			CNC_ZeroOffsets:
				IF (nLogChannelID <= 0 OR nLogChannelID > nLogChannelID) THEN
					nErrorID 	:= ErrID_7;
					Step := 999;
				ELSE
					Step := 12;
				END_IF
		END_CASE
	END_IF

	fbFileOpen.bExecute := FALSE;
	
	// Check Channel State
	IF (CNCSystem.LogChannelNo[nLogChannelID].nHliChannelIdx <> -1) THEN
		
		IF (cncSystem.Channel[CNCSystem.LogChannelNo[nLogChannelID].nHliChannelIdx].ActState <> HLI_IMCM_PROCESS_SELECTED AND 
			cncSystem.Channel[CNCSystem.LogChannelNo[nLogChannelID].nHliChannelIdx].ActState <> HLI_IMCM_PROCESS_READY) THEN
			nErrorID 	:= ErrID_10;
			Step := 999;
		END_IF				
	ELSE
			nErrorID 	:= ErrID_7;
			Step := 999;		
	END_IF			

12:	(* create file name and list file header  *)
	strHeader := '';

	CASE eParameterType OF

		CNC_AxisParameter:
			strFileName := CONCAT(strTempPath, '\axis');
			strFileName := CONCAT(strFileName, UINT_TO_STRING(nLogAxisId));
			strFileName := CONCAT(strFileName, '.lis');

			strHeader := 'kopf.achs_nr ';
			strHeader := CONCAT(strHeader, UINT_TO_STRING(nLogAxisId));
			Step := 15;
		CNC_ChannelParameter:
			strFileName := CONCAT(strTempPath, '\channel');			
			strFileName := CONCAT(strFileName, UINT_TO_STRING(nLogChannelID));
			strFileName := CONCAT(strFileName, '.lis');
			Step := 15;
		CNC_ToolParameter:			
			strFileName := CONCAT(strTempPath, '\ToolCh');
			strFileName := CONCAT(strFileName, UINT_TO_STRING(nLogChannelID));
			strFileName := CONCAT(strFileName, '.lis');
			Step := 15;
		CNC_ClampPosition:
			strFileName := CONCAT(strTempPath, '\ClampPosCh');			
			strFileName := CONCAT(strFileName, UINT_TO_STRING(nLogChannelID));
			strFileName := CONCAT(strFileName, '.lis');
			Step := 15;
		CNC_ZeroOffsets:			
			strFileName := CONCAT(strTempPath, '\ZeroOffsetsChh');
			strFileName := CONCAT(strFileName, UINT_TO_STRING(nLogChannelID));
			strFileName := CONCAT(strFileName, '.lis');
			Step := 15;
		ELSE
			nErrorID 	:= ErrID_5;
			Step := 999;
	END_CASE

15:	(* write file to destination folder *)
	fbFileOpen.sNetId := '';
	fbFileOpen.sPathName := strFileName;
	fbFileOpen.nMode := FOPEN_MODEWRITE OR FOPEN_MODETEXT;
	fbFileOpen.ePath := PATH_GENERIC;
	fbFileOpen.tTimeout := t#1s;
	fbFileOpen.bExecute := TRUE;
	Step := 16;

16:
	IF ( NOT fbFileOpen.bBusy ) THEN
		IF ( fbFileOpen.bError ) THEN
			nErrorID  :=ErrID_9 ;
			bError := TRUE;
			Step := 999;
		ELSE
			hFileOutput := fbFileOpen.hFile;
			fbFilePuts.bExecute:= FALSE;
			Step := 17;
		END_IF
	END_IF


17: (* Write Header File *)
	fbFilePuts.sNetId:='';
	fbFilePuts.hFile:=hFileOutput;
	fbFilePuts.bExecute:=TRUE;
	fbFilePuts.tTimeout:=t#10s;
	fbFilePuts.sLine :=strHeader;
	Step := 18;

18:
	IF ( NOT fbFilePuts.bBusy ) THEN
		IF ( fbFilePuts.bError ) THEN
			 nErrorID  :=ErrID_9 ;
			bError := TRUE;
			Step := 999;
		ELSE
			fbFilePuts.bExecute:= FALSE;
			m := 0;
			Step := 19;
		END_IF
	END_IF


19:	(* Write Parameter lines *)
		strParameterLine :=  CONCAT('$N',stParameter[m].strName);
		strParameterLine :=  CONCAT(strParameterLine,'   ');
		strParameterLine := CONCAT(strParameterLine, stParameter[m].strValue);
		fbFilePuts.sLine :=strParameterLine;
		fbFilePuts.bExecute:= TRUE;
		Step := 20;
20:
		IF ( NOT fbFilePuts.bBusy ) THEN
			IF ( fbFilePuts.bError ) THEN
				 nErrorID  :=ErrID_9 ;
				bError := TRUE;
				Step := 999;
			ELSE
				Step := 21;
			END_IF
		END_IF

21:	(* Next Line *)
	IF (m+1 <= (nMaxParameters-1) AND m+1 <= nNumParameters) THEN
		m := m+1;
		fbFilePuts.bExecute:= FALSE;
		Step := 19;
	ELSE
		fbFilePuts.bExecute:= FALSE;
		Step := 22;
	END_IF

22:	(* Write footer *)
	fbFilePuts.sLine :='$NEnde';
	fbFilePuts.bExecute:= TRUE;
	Step := 23;

23:
	IF ( NOT fbFilePuts.bBusy ) THEN
		IF ( fbFilePuts.bError ) THEN
			 nErrorID  :=ErrID_9 ;
			bError := TRUE;
			Step := 999;
		ELSE
			fbFileClose.bExecute:=FALSE;
			Step := 30;
		END_IF
	END_IF


30:	(* Close File *)
	fbFileClose.sNetId:='';
	fbFileClose.hFile:=hFileOutput;
	fbFileClose.bExecute:=TRUE;
	fbFileClose.tTimeout:=t#1s;

	IF ( NOT fbFileClose.bBusy ) THEN
		IF ( fbFileClose.bError ) THEN
			 nErrorID  :=ErrID_9 ;
			bError := TRUE;
			Step := 999;
		ELSE
			hFileOutput := 0;
			Step := 35;
		END_IF
	END_IF

	35:
		CASE eParameterType OF
			CNC_AxisParameter:
				Step := 60;
			CNC_ChannelParameter:
				Step := 60;
			CNC_ToolParameter:
				Step := 60;
			CNC_ClampPosition:
				Step := 60;
			CNC_ZeroOffsets:
				Step := 60;
		END_CASE

	40:	(* logical axis ID*)
		TimeOut(IN:=FALSE);
		FbAdsWrite( Port := 553, IdxGrp := nAdsIndexGroup  + nLogChannelID, IdxOffs := (nAdsIndexOffsetlogAxisNumber), LEN := SIZEOF(nLogAxisID), SrcAddr := ADR(nLogAxisID),TMOUT := T#1S, WRITE := TRUE);
		Step := 50;
	50:
		TimeOut(IN:=TRUE, PT:=T#2S);

		FbAdsWrite();
		IF FbAdsWrite.BUSY = FALSE THEN
			IF NOT FbAdsWrite.ERR THEN
				FbAdsWrite( WRITE := FALSE);
				Step := 60;
			ELSE
				FbAdsWrite( WRITE := FALSE);
				nErrorID := ErrID_3;
				Step := 999;
			END_IF
		END_IF

		(* error timeout *)
		IF TimeOut.Q THEN
			nErrorID 	:= ErrID_1;
			Step   	:= 999;
		END_IF

	60:	(* activate List File *)
		TimeOut(IN:=FALSE);

		CASE eParameterType OF

		CNC_AxisParameter:
			FbAdsWrite( Port := nAdsPortNumber, IdxGrp := nAdsIndexGroupAxisParameter  + nLogAxisId, IdxOffs := (nAdsIndexOffsetAxisParameter), LEN := SIZEOF(strFileName), SrcAddr := ADR(strFileName), WRITE := TRUE);
		CNC_ChannelParameter:
			FbAdsWrite( Port := nAdsPortNumber, IdxGrp := nAdsIndexGroup  + nLogChannelID, IdxOffs := (nAdsIndexOffsetChannelParameter), LEN := SIZEOF(strFileName), SrcAddr := ADR(strFileName), WRITE := TRUE);
		CNC_ToolParameter:
			FbAdsWrite( Port := nAdsPortNumber, IdxGrp := nAdsIndexGroup  + nLogChannelID, IdxOffs := (nAdsIndexOffsetToolParameter), LEN := SIZEOF(strFileName), SrcAddr := ADR(strFileName), WRITE := TRUE);
		CNC_ClampPosition:
			FbAdsWrite( Port := nAdsPortNumber, IdxGrp := nAdsIndexGroup  + nLogChannelID, IdxOffs := (nAdsIndexOffsetClampPosition), LEN := SIZEOF(strFileName), SrcAddr := ADR(strFileName), WRITE := TRUE);
		CNC_ZeroOffsets:
			FbAdsWrite( Port := nAdsPortNumber, IdxGrp := nAdsIndexGroup  + nLogChannelID, IdxOffs := (nAdsIndexOffsetZeroOffsets), LEN := SIZEOF(strFileName), SrcAddr := ADR(strFileName), WRITE := TRUE);
		END_CASE

		Step := 70;
	70:
		TimeOut(IN:=TRUE, PT:=T#2S);
		FbAdsWrite();
		IF FbAdsWrite.BUSY = FALSE THEN

			IF NOT FbAdsWrite.ERR THEN
				FbAdsWrite( WRITE := FALSE);
				Step := 0;
			ELSE
				FbAdsWrite( WRITE := FALSE);
				nErrorID := ErrID_4;
				Step := 999;
			END_IF
		END_IF

		(* error timeout *)
		IF TimeOut.Q THEN
			nErrorID 	:= ErrID_1;
			Step   	:= 999;
		END_IF

999: (* Fehler *)
		bBusy  := FALSE;
		bError := TRUE;
		Step 	 := 0;
END_CASE

fbFileOpen();
fbFilePuts();
fbFileClose();

END_FUNCTION_BLOCK

// CNC/11 Util/FB_Uint_Udint
FUNCTION_BLOCK FB_Uint_Udint
VAR
	nOldValue: UINT;
	nDiff: DINT;
	nMinus: BOOL;
	nPlus: BOOL;
END_VAR
VAR_INPUT
	nInSmall: UINT;
END_VAR

VAR_IN_OUT
	nBig: UDINT;
END_VAR

nDiff := nInSmall - nOldValue;


(* Richtung Minus *)
IF ndiff > 10000 THEN
	nBig := nBig - 1;
	nMinus := TRUE;
END_IF

(* Richtung Plus *)
IF ndiff < -10000 THEN
	nBig := nBig + 1;
	nPlus := TRUE;
END_IF

IF (ndiff < 500) AND ndiff > -500 THEN
  nBig := DINT_TO_UDINT( UDINT_TO_DINT(nBig) + nDiff) ;
END_IF
nOldValue := nInSmall;

END_FUNCTION_BLOCK

// CNC/11 Util/HLI3_FindAxisNameAndChannel
FUNCTION HLI3_FindAxisNameAndChannel : BOOL
VAR_INPUT
	LogAxeNr		: UDINT;
	pAxisName		: POINTER TO STRING(HLI_ACHS_NAME_LAENGE);
	pChannelNr		: POINTER TO UINT;
END_VAR
VAR
	i				: UDINT;
	
	pString			: POINTER TO STRING;
END_VAR

FOR i := 0 TO gNrAx - 1 DO
	IF gpAx[i]^.ipo_state.log_achs_nr_r = LogAxeNr THEN
		pChannelNr^ := gpAx[i]^.ipo_state.cnc_channel_r;	(* channel of axis *)
		FOR i := 0 TO INT_TO_UDINT(HLI_CH_AX_MAXIDX) DO
			IF gpCh[pChannelNr^-1]^.bahn_state.coord_r[i].log_achs_nr_r = LogAxeNr THEN
				pString                := ADR(gpCh[pChannelNr^-1]^.bahn_state.coord_r[i].axis_name_r.zeichen);	(* name of axis *)
				pAxisName^             := pString^;
				HLI3_FindAxisNameAndChannel := TRUE;
				RETURN;
			END_IF
		END_FOR
	END_IF
END_FOR

pAxisName^ := '';
pChannelNr^ := 0;
HLI3_FindAxisNameAndChannel := FALSE;

END_FUNCTION

// CNC/11 Util/HLI3_FindHliAxisIdx
FUNCTION HLI3_FindHliAxisIdx : DINT
VAR_INPUT
	nLogAxisNo		: UDINT;	
END_VAR
VAR
	i				: UINT;	
END_VAR

IF nLogAxisNo > MAX_SYS_LOG_AXIS_INDEX OR nLogAxisNo < 1 THEN 
	HLI3_FindHliAxisIdx := -1;
ELSE
	HLI3_FindHliAxisIdx := CNCSystem.LogAxisNo[nLogAxisNo].nHliAxisIdx;	
END_IF

END_FUNCTION

// CNC/11 Util/HLI3_GetEtherCATAxisInfo
FUNCTION HLI3_GetEtherCATAxisInfo : ST_DriveRef
VAR
	arrTemp: ARRAY[1..24] OF BYTE;
	arrNetIdAchse2: ARRAY[0..MAX_STRING_LENGTH] OF BYTE;
	i: INT;
	id: DINT;
	nCha: UINT;
	nPort: UINT;
END_VAR
VAR_INPUT
	nHliAxisIdx: INT;
END_VAR

(* ========================================================= *)
(*    FUN: HLI_GetEtherCATAxisInfo                   		 *)
(* --------------------------------------------------------- *)
(*   Desc: Gets the information about a SoE Drive (Ax5000)   *)
(*  benötigt: TcEtherCAT.lib   *)
(* Return: Structure with the information for the drive     *)
(* Author: MiB                                               *)
(*   Date: 20.11.2012                                        *)
(*   Rev.: 1.2                                               *)
(* ========================================================= *)


IF NOT HLI3_CheckAxisValid(nHliAxisIdx := nHliAxisIdx) THEN
	HLI3_GetEtherCATAxisInfo.sNetId := '';
	HLI3_GetEtherCATAxisInfo.nDriveNo := 0;
	HLI3_GetEtherCATAxisInfo.nSlaveAddr := 0;
	RETURN;	
END_IF


HLI3_GetEtherCATAxisInfo.sNetId := gpAx[nHliAxisIdx]^.lr_state.twincat_box.ads_netid_r;
HLI3_GetEtherCATAxisInfo.nDriveNo := UINT_TO_BYTE(gpAx[nHliAxisIdx]^.lr_state.twincat_box.channel_r);
HLI3_GetEtherCATAxisInfo.nSlaveAddr :=gpAx[nHliAxisIdx]^.lr_state.twincat_box.ads_port_r;

RETURN;

END_FUNCTION

// CNC/11 Util/HLI3_SoftwareLimitSwitches
///*********************************************************************************************************
///NAME.......................:		HLI3_SoftwareLimitSwitches
///DATUM....................:		22.12.2017
///AUTOR....................:		Thomas Voß
///VERSION................:			1.1
///
///Description.: 	Read and Write Software Limit Switches					
///**********************************************************************************************************

FUNCTION_BLOCK HLI3_SoftwareLimitSwitches
VAR_INPUT
	nChannelId		: UINT;
	nLogAxisId		: UINT;	
	fSWLimitNeg		: LREAL;
	fSWLimitPos		: LREAL;
	bExecute		: BOOL;
	/// Windows temp file for sub lists
	strTempPath: STRING;
END_VAR
VAR_OUTPUT
	bBusy  : BOOL;
	bError : BOOL;
	ErrID  :  INT;
END_VAR
VAR
	fbOnTrigger		:  	R_TRIG;

	Step 			: 	UDINT;
		/// Text To File 
	fbFileOpen		: 	FB_FileOpen;
	fbFileRead		: 	FB_FileRead;
	fbFilePuts		: 	FB_FilePuts;
	fbFileClose		: 	FB_FileClose;
	hFileOutput		: 	UINT := 0;
	FbAdsWrite		: 	ADSWRITE;
	FbAdsRead		: 	ADSREAD;
	text			:	STRING(255);
	file			:	STRING(255);
	nSETSWLimitNegValue	: DINT;
	nSETSWLimitPosValue	: DINT;
	Get_SWLimitNeg 	: 	DINT;
	Get_SWLimitPos  : 	DINT;
	offset 			: 	UDINT;
	TimeOut 		: 	TON;	
END_VAR

VAR CONSTANT
	ErrID_1:								INT := 1;		(* Time Out Error *)
	ErrID_2:								INT := 2;		(* Fehler beim Öffnen der Parameterdatei *)
	ErrID_3:								INT := 3;		(* ADS - Fehler : Vorgabe Achs ID *)
	ErrID_4:								INT := 4;		(* ADS - Fehler : Aktivierung der Parameterliste *)
	ErrID_5:								INT := 5;		(* ADS - Fehler :Fehler beim Lesen vom negativen Endschalter  *)
	ErrID_6:								INT := 6;		(* ADS - Fehler :Fehler beim Lesen vom positiven Endschalter  *)
	ErrID_7:								INT := 7;		(* Fehler : Set - SW Limit Switch <> Get SW Limit Switch   *)
	ErrID_9:								INT := 9;		(* File Write Error *)
	ErrID_10:								INT := 10;		(* Invalid AxisId *)
	ErrID_11:								INT := 11;		(* Invalid Limit Parameters *)
	ErrID_12:								INT := 12;		(* No File Path configured*)
	ErrID_13:								INT := 13;		(* Invalid ChannelId *)
END_VAR

fbOnTrigger(CLK:= bExecute);

IF fbOnTrigger.Q THEN
	Step 	:= 10;
	ErrID 	:= 0;
	bError	 := 0;
	bBusy := TRUE;
END_IF

CASE Step OF
0:
	bBusy := FALSE;

10:		// Check Input Parameters 
		nSetSWLimitNegValue	:= LREAL_TO_DINT(fSWLimitNeg*10000);
		nSetSWLimitPosValue	:= LREAL_TO_DINT(fSWLimitPos*10000);
		
		IF (nLogAxisId < 0) THEN
			bError :=	TRUE;
			ErrID  :=  ErrID_10;
			Step   := 999;
		ELSIF  (nLogAxisId > MAX_SYS_LOG_AXIS_INDEX) THEN
			bError :=	TRUE;
			ErrID  :=  ErrID_10;
			Step   := 999;
		ELSIF (CNCSystem.LogAxisNo[nLogAxisId].nHliAxisIdx = -1) THEN
			bError :=	TRUE;
			ErrID  :=  ErrID_10;
			Step   := 999;
		ELSIF (nSETSWLimitNegValue > nSetSWLimitPosValue) OR (nSETSWLimitNegValue = nSetSWLimitPosValue) THEN	
			bError :=	TRUE;
			ErrID  :=   ErrID_11;
			Step   :=   999;
		ELSIF (strTempPath = '') THEN
			bError :=	TRUE;
			ErrID  :=   ErrID_12;
			Step   :=   999;
		ELSIF (nChannelId < 1 OR UINT_TO_INT(nChannelId) > HLI_SYS_CH_MAXIDX+1) THEN
			bError :=	TRUE;
			ErrID  :=   ErrID_13;
			Step   :=   999; 
		ELSE
			Step 	:= 20;		
		END_IF		
					
20:
		file := CONCAT(strTempPath, '\axis');
		file := CONCAT(file, UINT_TO_STRING(nLogAxisId));
		file := CONCAT(file, '.lis');
								
		text := 'kopf.achs_nr ';
		text := CONCAT(text, UINT_TO_STRING(nLogAxisId));
		text := CONCAT(text, '$Nkenngr.swe_neg    ');
		text := CONCAT(text, DINT_TO_STRING(nSetSWLimitNegValue));
		text := CONCAT(text, '$Nkenngr.swe_pos    ');
		text := CONCAT(text, DINT_TO_STRING(nSetSWLimitPosValue));
		text := CONCAT(text, '$NEnde');

		TimeOut(IN:=FALSE);
		fbFileOpen.bExecute := FALSE;
		Step := Step+10;
					
30:	(* write file to destination folder *)
	fbFileOpen.sNetId := '';
	fbFileOpen.sPathName := file;
	fbFileOpen.nMode := FOPEN_MODEWRITE OR FOPEN_MODETEXT;
	fbFileOpen.ePath := PATH_GENERIC;
	fbFileOpen.tTimeout := t#1s;
	fbFileOpen.bExecute := TRUE;
	Step := Step+10;

40:
	IF ( NOT fbFileOpen.bBusy ) THEN
		IF ( fbFileOpen.bError ) THEN
			ErrID  :=ErrID_9 ;
			bError := TRUE;
			Step := 999;
		ELSE
			hFileOutput := fbFileOpen.hFile;
			fbFilePuts.bExecute:= FALSE;
			Step := Step+10;
		END_IF
	END_IF

50: (* Write Header File *)
	fbFilePuts.sNetId:='';
	fbFilePuts.hFile:=hFileOutput;
	fbFilePuts.bExecute:=TRUE;
	fbFilePuts.tTimeout:=t#10s;
	fbFilePuts.sLine :=text;
	Step := Step+10;

60:
	IF ( NOT fbFilePuts.bBusy ) THEN
		IF ( fbFilePuts.bError ) THEN
			ErrID  :=ErrID_9 ;
			bError := TRUE;
			Step := 999;
		ELSE
			fbFilePuts.bExecute:= FALSE;		
			Step := Step+10;
		END_IF
	END_IF

70:
	IF ( NOT fbFilePuts.bBusy ) THEN
		IF ( fbFilePuts.bError ) THEN
			ErrID  :=ErrID_9 ;
			bError := TRUE;
			Step := 999;
		ELSE
			fbFileClose.bExecute:=FALSE;
			Step := Step+10;
		END_IF
	END_IF


80:	(* Close File *)
	fbFileClose.sNetId:='';
	fbFileClose.hFile:=hFileOutput;
	fbFileClose.bExecute:=TRUE;
	fbFileClose.tTimeout:=t#1s;

	IF ( NOT fbFileClose.bBusy ) THEN
		IF ( fbFileClose.bError ) THEN
			ErrID  :=ErrID_9 ;
			bError := TRUE;
			Step := 999;
		ELSE
			hFileOutput := 0;
			Step := Step+10;
		END_IF
	END_IF
		
90:		(* logical axis ID*)
		TimeOut(IN:=FALSE);
		FbAdsWrite( Port := 553, IdxGrp := 16#20100 + nChannelId, IdxOffs := (16#37), LEN := SIZEOF(nLogAxisId), SrcAddr := ADR(nLogAxisId),TMOUT := T#1S, WRITE := TRUE);
		Step := Step+10;
100:
		TimeOut(IN:=TRUE, PT:=T#2S);

		FbAdsWrite();
		IF FbAdsWrite.BUSY = FALSE THEN
			IF NOT FbAdsWrite.ERR THEN
				FbAdsWrite( WRITE := FALSE);
				Step := Step+10;
			ELSE
				FbAdsWrite( WRITE := FALSE);
				ErrID := ErrID_3;
				Step := 999;
			END_IF
		END_IF

		(* error timeout *)
		IF TimeOut.Q THEN
			ErrID 	:= ErrID_1;
			Step   	:= 999;
		END_IF

110:		(* Achsparameter aktivieren *)
		TimeOut(IN:=FALSE);

	    FbAdsWrite( WRITE := FALSE);
		FbAdsWrite( Port := 553, IdxGrp := 16#20100 + nChannelId, IdxOffs := (16#36), LEN := SIZEOF(file), SrcAddr := ADR(file), WRITE := TRUE);
		Step := Step+10;
		
120:
		TimeOut(IN:=TRUE, PT:=T#2S);
		FbAdsWrite();
		IF FbAdsWrite.BUSY = FALSE THEN

			IF NOT FbAdsWrite.ERR THEN
				FbAdsWrite( WRITE := FALSE);
				FbAdsRead(Read:=FALSE);
				Step := Step+10;
			ELSE
				FbAdsWrite( WRITE := FALSE);
				ErrID := ErrID_4;
				Step := 999;
			END_IF
		END_IF

		(* error timeout *)
		IF TimeOut.Q THEN
			ErrID 	:= ErrID_1;
			Step   	:= 999;
		END_IF

130: (* Read negative Limit Switch *)
	TimeOut(IN:=FALSE);
	FbAdsRead(	NETID:= '',				(* local *)
				PORT:= 553,					(* Port number of Task COM, all ADS-Requests to the NC-kernel  *)										(* must sent to this port                                      *)
				IDXGRP:=16#00020200+nLogAxisId,    (*  *)
				IDXOFFS:= 16#26,
				LEN:=SIZEOF(Get_SWLimitNeg),		(* number of bytes that shall be read                          *)
				DESTADDR:= ADR(Get_SWLimitNeg),  (* memory for the read value, must be provided by the user     *)
				READ:=TRUE,					(* a rising edge on this input starts the read request         *)
				TMOUT:= T#1s);       (* maximum time for read request                               *)

		Step := Step+10;

140:
		TimeOut(IN:=TRUE, PT:=T#2S);
		FbAdsRead();
		IF NOT FbAdsRead.Busy THEN
			IF NOT FbAdsRead.ERR THEN
				FbAdsRead(READ := FALSE);
				Step := Step+10;
			ELSE
				FbAdsRead(READ := FALSE);
				ErrID 	:= ErrID_5;
				Step := 999;
			END_IF
		END_IF

		(* error timeout *)
		IF TimeOut.Q THEN
			ErrID 	:= ErrID_1;
			Step   	:= 999;
		END_IF



150: (* Read positive Limit Switch *)
	TimeOut(IN:=FALSE);
	FbAdsRead(	NETID:= '',				(* local *)
				PORT:= 553,					(* Port number of Task COM, all ADS-Requests to the NC-kernel  *)										(* must sent to this port                                      *)
				IDXGRP:=16#00020200+nLogAxisId,    (*  *)
				IDXOFFS:= 16#25,
				LEN:=SIZEOF(Get_SWLimitPos),		(* number of bytes that shall be read                          *)
				DESTADDR:= ADR(Get_SWLimitPos),  (* memory for the read value, must be provided by the user     *)
				READ:=TRUE,					(* a rising edge on this input starts the read request         *)
				TMOUT:= T#1s);       (* maximum time for read request                               *)
	Step := Step+10;

160:	TimeOut(IN:=TRUE, PT:=T#2S);
		FbAdsRead();
		IF NOT FbAdsRead.Busy THEN
			IF NOT FbAdsRead.ERR THEN
				FbAdsRead(READ := FALSE);
				Step := Step+10;
			ELSE
				FbAdsRead(READ := FALSE);
				ErrID 	:= ErrID_6;
				Step := 999;
			END_IF
		END_IF

170:	(* Check *)
		IF (Get_SWLimitNeg = nSetSWLimitNegValue) AND (Get_SWLimitPos = nSetSWLimitPosValue) THEN
			bBusy := FALSE;
			Step := 0;
		ELSE
			ErrID 	:= ErrID_7;
			Step := 999;
		END_IF


999: (* Fehler *)
		bBusy  := FALSE;
		bError := TRUE;
		Step 	 := 0;
END_CASE

fbFileOpen();
fbFilePuts();
fbFileClose();

END_FUNCTION_BLOCK

// CNC/12 CNC_Axis/FB_ActivateCompTable
(**********************************************************************************************************
NAME...................:		FB_ActivateSSFK	
DATUM..................:		23.01.2009
AUTOR..................:		Thomas Voß
VERSION................:		1.0

BESCHREIBUNG.:	Aktiviert Korrekturwerttabelle über den CNC List File Interpreter
......................: 	

***********************************************************************************************************)
FUNCTION_BLOCK FB_ActivateCompTable
VAR_INPUT
	bExecute			: BOOL;
	strPathCompTable 	: STRING(256);
	nAxisID				: DINT;
	tTimeout			: TIME := T#10S;
END_VAR
VAR_OUTPUT
	bBusy			: 	BOOL;
	bError			:	BOOL;
	nErrID			:	UDINT;
END_VAR
VAR
	iState 			:  UINT;
	fbOnTrigger		:  R_TRIG;
	fbAdsWrite		:  ADSWRITE;
END_VAR

fbOnTrigger(CLK:= bExecute);

CASE iState OF

0 :

	bBusy := FALSE;

	IF fbOnTrigger.Q THEN
			iState := 10;
			nErrID := 0;
			bError := 0;
			bBusy := TRUE;
			fbAdsWrite(WRITE := FALSE);
		END_IF


10:                (* logical axis ID*)
                fbAdsWrite( Port := 553, IdxGrp := 16#20101, IdxOffs := (16#3A), LEN := SIZEOF(nAxisID), SrcAddr := ADR(nAxisID), WRITE := TRUE);

		IF NOT fbAdsWrite.Busy THEN
			IF fbAdsWrite.Err THEN
				bError := fbAdsWrite.Err;
				nErrID :=fbAdsWrite.ERRID;
				iState := 0;
			ELSE
				fbAdsWrite(WRITE := FALSE);
				iState := 20;
			END_IF
		END_IF


20: (* Korrekturwert Tabelle aktivieren *)

                FbAdsWrite( Port := 553, IdxGrp := 16#20101, IdxOffs := (16#39), LEN := SIZEOF(strPathCompTable), SrcAddr := ADR(strPathCompTable), WRITE := TRUE);

		IF NOT fbAdsWrite.Busy THEN
			IF fbAdsWrite.Err THEN
				bError := fbAdsWrite.Err;
				nErrID :=fbAdsWrite.ERRID;
				iState := 0;
			ELSE
				fbAdsWrite(WRITE := FALSE);
				iState := 0;
			END_IF
		END_IF

END_CASE

END_FUNCTION_BLOCK

// CNC/12 CNC_Axis/FB_CNCAxis
FUNCTION_BLOCK FB_CNCAxis EXTENDS HLI3_CNCAxisBase
VAR_INPUT
	nLogAxisNo : INT;
END_VAR
VAR_OUTPUT
END_VAR
VAR
END_VAR

(* ========================================================= *)
(*     FB: FB_CNCAxis                                  		 *)
(* --------------------------------------------------------- *)
(*   Desc:  CNC Axis Control							   	 *)
(*   Author: TV				                                 *)
(*   Date: 2018.01.25                                        *)
(*   Rev.: 1.0                                               *)
(* ==========================================================*)

IF nLogAxisNo < 1 OR  nLogAxisNo > UINT_TO_INT(MAX_SYS_LOG_AXIS_INDEX) THEN
	RETURN;
END_IF

IF CNCSystem.LogAxisNo[nLogAxisNo].nHliAxisIdx = -1 THEN
	RETURN;
END_IF

SUPER^(nHliIdx := CNCSystem.LogAxisNo[nLogAxisNo].nHliAxisIdx);

END_FUNCTION_BLOCK

// CNC/12 CNC_Axis/HLI3_CNCAxisBase
FUNCTION_BLOCK HLI3_CNCAxisBase
VAR_INPUT
	{attribute 'hide'}
	nHliIdx						: INT;
	bEnable 					: BOOL;	
  //  bEnablePositive 			: BOOL; 
  //  bEnableNegative 			: BOOL; 
	bCalibrationCam				: BOOL;		
	bSetRefOffset				: BOOL;
	fRefOffset					: LREAL;  // [ mm or degree ] 	
	stOptions           		: ST_CNC_AX_Options;	
	stParameter					: ST_CNC_AX_Parameter;
	stPLCopen					: ST_CNC_AX_PLCopen;
END_VAR
VAR_OUTPUT
	stStatus					: ST_CNC_AX_Status;	
END_VAR
VAR
	fbSetAxisRelease 			: HLI3_SetAxisRelease;
	fbSetAxisReferenceOffset	: HLI3_SetAxisReferenceOffset;
	fbActivateCompTable			: FB_ActivateCompTable;
	bInit 						: BOOL;
	fbOnTrigger					: R_TRIG;
	nStepWriteParam				: INT;
	fbOnTriggerCompTable		: R_TRIG;
	nStepActivateCompTable      : INT;
	
	// PLCopen Platform
	fbMC_SetOverride			: MC_SetOverride;
	fbMC_Home					: MC_Home;
	fbMC_MoveAbsolute			: MC_MoveAbsolute;
	fbMC_ReadAxisError 			: MC_ReadAxisError;	
	fbMC_Stop					: MC_Stop;
	fbMC_Reset					: MC_Reset;
END_VAR

(* ========================================================= *)
(*     FB: FB_CNCAxis                                  		 *)
(* --------------------------------------------------------- *)
(*   Desc:  CNC Axis Control							   	 *)
(*   Author: TV				                                 *)
(*   Date: 2018.03.19                                        *)
(*   Rev.: 1.4                                               *)
(* ==========================================================*)

IF NOT CNCSystem.bHLIInit THEN
	RETURN;
END_IF

IF NOT (HLI3_CheckAxisValid(nHliAxisIdx := nHliIdx)) THEN
	RETURN;
END_IF

ACT_Init();
ACT_Parameter();
ACT_Status();
ACT_Options();
ACT_PLCopen();

// Axis Release
fbSetAxisRelease(
	bEnable:= bEnable, 
	nHliAxisIdx:= nHliIdx);
	
// Reference Cam        
HLI3_SetAxisReferenceCam(nHliIdx,bCalibrationCam);

// Set Ref. Offset
fbSetAxisReferenceOffset(
	Execute:= bSetRefOffset, 
	nHliAxisIdx:= nHliIdx, 
	nOffset:= fRefOffset);

ACTION ACT_Init:
IF NOT bInit THEN
	gpAX[nHliIdx]^.ipo_mc_control.reduced_speed.enable_w := TRUE;
	gpAX[nHliIdx]^.ipo_mc_control.reduced_speed_zone.enable_w := TRUE;
	gpAX[nHliIdx]^.ipo_mc_control.reduced_speed_2_zone.enable_w := TRUE;
END_IF
END_ACTION

ACTION ACT_Options:
// Clear Reference Position
HLI3_ClearReferencePosition(nHliAxisIdx := nHliIdx, bExecute := stOptions.bResetCalibration);

// Probing Signal       
HLI3_SetProbingSignal(nHliIdx,stOptions.bProbingSignal);

// Reduced_Speed
gpAX[nHliIdx]^.ipo_mc_control.reduced_speed.command_w := stOptions.bReducedSpeed;

// Reduced_Speed Zone 1
gpAX[nHliIdx]^.ipo_mc_control.reduced_speed_zone.command_w := stOptions.bReducedSpeedZone1;

// Reduced_Speed Zone 2
gpAX[nHliIdx]^.ipo_mc_control.reduced_speed_2_zone.command_w := stOptions.bReducedSpeedZone2;
 
// Activate Compensation Table
fbOnTriggerCompTable(CLK:= stOptions.bActivateCompTable);

IF fbOnTriggerCompTable.Q THEN
	nStepActivateCompTable:= 10;
END_IF

CASE nStepActivateCompTable OF
0:

10:
	IF NOT fbActivateCompTable.bBusy AND NOT bCNC_AX_ActivateCompTableLock  THEN
			bCNC_AX_ActivateCompTableLock  := TRUE;						 
			fbActivateCompTable.bExecute:= FALSE;	 
			nStepActivateCompTable := 20;	
	END_IF	
20:			
	fbActivateCompTable.bExecute:= TRUE;
    fbActivateCompTable.strPathCompTable:= stOptions.strPathCompTable; 
	fbActivateCompTable.nAxisID:= gpAx[nHliIdx]^.head.log_ax_nr_r;	
	nStepActivateCompTable := 30;			 				
	
30:	IF NOT fbActivateCompTable.bBusy OR  fbActivateCompTable.bError THEN		
		bCNC_AX_ActivateCompTableLock := FALSE;
		nStepActivateCompTable := 0;		
	END_IF
	
END_CASE
END_ACTION

ACTION ACT_Parameter:


fbOnTrigger(CLK:= stParameter.bWriteParameter);

IF fbOnTrigger.Q THEN
	nStepWriteParam := 10;
END_IF

CASE nStepWriteParam OF
0:

10:
	IF NOT fbCNC_AX_WriteParameter.bBusy AND NOT bCNC_AX_WriteParameterLock THEN
			bCNC_AX_WriteParameterLock := TRUE;						 
			fbCNC_AX_WriteParameter.bExecute:= FALSE;	 
			nStepWriteParam := 20;	
	END_IF
	
20:			 
			fbCNC_AX_WriteParameter.nLogChannelID:= 1;		 
			fbCNC_AX_WriteParameter.nLogAxisId:= gpAx[nHliIdx]^.head.log_ax_nr_r; 
			fbCNC_AX_WriteParameter.bExecute:= TRUE; 
			fbCNC_AX_WriteParameter.nNumParameters:= stParameter.nNumParameters;
			fbCNC_AX_WriteParameter.eParameterType:= E_CNCParameterTypes.CNC_AxisParameter; 
			fbCNC_AX_WriteParameter.strTempPath:= stParameter.strTempPath; 		 
			fbCNC_AX_WriteParameter.stParameter:= stParameter.ParamList;
			nStepWriteParam := 30;	
	
30:	IF NOT fbCNC_AX_WriteParameter.bBusy OR  fbCNC_AX_WriteParameter.bError THEN		
		bCNC_AX_WriteParameterLock:= FALSE;
		nStepWriteParam := 0;		
	END_IF
	
END_CASE
END_ACTION

ACTION ACT_PLCopen:
IF 	CNCSystem.bPLCopenPlatformInit AND 
	gpAx[nHliIdx]^.lr_state.is_sai_r AND
	g_array_axis_ref[nHliIdx].axsd_state <> MCV_AXSD_STATES.INIT_STATE	
THEN

(* Override *)
IF stPLCopen.nOverride > 1000 THEN stPLCopen.nOverride := 1000; END_IF  
IF stPLCopen.nOverride < 0 THEN stPLCopen.nOverride := 0; END_IF

fbMC_SetOverride(
	Axis:= g_array_axis_ref[nHliIdx],  
	Enable:= TRUE, 
	VelFactor:= UINT_TO_LREAL(stPLCopen.nOverride) / 1000.0, 
	VelFactorMaxShift:= , 
	Enabled=> , 
	Error=> , 
	ErrorID=> );
	
fbMC_Home(
	Axis:= g_array_axis_ref[nHliIdx], 
	Execute:= stPLCopen.bExecuteHoming, 
	CamSignal:= stPLCopen.bCamSignal,
	Done=> stStatus.PLCopen.bHomingDone,
	CommandAborted=> , 
	Error=> , 
	ErrorID=> );	
	
fbMC_MoveAbsolute(
	Axis:= g_array_axis_ref[nHliIdx], 
	Execute:=  stPLCopen.bExecuteMoveAbsolute, 
	Position:= stPLCopen.fPosition * 10000.0, 
	Velocity:= stPLCopen.fVelocity * 16.6666,
	Acceleration:= stPLCopen.fAcceleration, 
	Deceleration:= stPLCopen.fAcceleration,
	Jerk:= stPLCopen.fJerk, 
	Direction:= , 
	Done=> stStatus.PLCopen.bMoveAbsoluteDone, 
	CommandAborted=> , 
	Error=> , 
	ErrorID=> );	
	
	
	fbMC_Stop(
	Axis:= g_array_axis_ref[nHliIdx],  
	Execute:= stPLCopen.bExecuteStop, 
	Deceleration:= stPLCopen.fAcceleration,  
	Jerk:= stPLCopen.fJerk,  
	Done=> stStatus.PLCopen.bStopDone, 
	Error=> , 
	ErrorID=> );
	
	fbMC_Reset(
	Axis:= g_array_axis_ref[nHliIdx], 
	Execute:= stPLCopen.bExecuteReset,  
	Done=> stStatus.PLCopen.bResetDone, 
	Error=> , 
	ErrorID=> );
				
	stStatus.PLCopen.bError := fbMC_SetOverride.Error OR fbMC_MoveAbsolute.Error OR fbMC_Home.Error OR fbMC_Stop.Error OR fbMC_Reset.Error;;

	IF fbMC_SetOverride.ErrorID <> 0 THEN 
		stStatus.PLCopen.nErrorID := fbMC_SetOverride.ErrorID;
	ELSIF fbMC_Reset.ErrorID <> 0 THEN 
		stStatus.PLCopen.nErrorID := fbMC_Reset.ErrorID;
	ELSIF fbMC_Stop.ErrorID <> 0 THEN
		stStatus.PLCopen.nErrorID := fbMC_Stop.ErrorID;
	ELSIF fbMC_Home.ErrorID <> 0 THEN 
		stStatus.PLCopen.nErrorID := fbMC_Home.ErrorID;
	ELSIF fbMC_MoveAbsolute.ErrorID <> 0 THEN  
		stStatus.PLCopen.nErrorID := fbMC_MoveAbsolute.ErrorID;		
	ELSE 		
		stStatus.PLCopen.nErrorID := 0;
	END_IF
	
	IF stStatus.PLCopen.nErrorID = 40001 THEN 
	
		fbMC_ReadAxisError(
			Axis:= g_array_axis_ref[nHliIdx],  
			Enable:= TRUE);
			
			IF fbMC_ReadAxisError.AxisErrorID <> 0 THEN
				stStatus.PLCopen.nErrorID := UDINT_TO_DINT(fbMC_ReadAxisError.AxisErrorID);
			END_IF
			
	END_IF
			
END_IF
END_ACTION

ACTION ACT_Status:
stStatus.bHomingDone := gpAx[nHliIdx]^.lr_state.homing_done_r;

stStatus.fSetPosACS	:= DINT_TO_LREAL(gpAx[nHliIdx]^.lr_state.active_position_acs_r) / 10000.0;;
stStatus.fActPosACS	:= DINT_TO_LREAL(gpAx[nHliIdx]^.lr_state.current_position_acs_r) / 10000.0;


IF (gpAx[nHliIdx]^.ipo_state.spindle_axis_r) THEN // Spindle
	stStatus.fActVelo := DINT_TO_LREAL( gpAx[nHliIdx]^.lr_state.current_rev_r) / 16.66666666 / 360.00;
ELSE
	stStatus.fActVelo := DINT_TO_LREAL( gpAx[nHliIdx]^.lr_state.current_rev_r) / 16.66666666;
END_IF

// CNC Axis Error ID
IF (gpAx[nHliIdx]^.ipo_state.cnc_channel_r > 0 ) THEN

	IF gpCh[CNCSystem.LogChannelNo[gpAx[nHliIdx]^.ipo_state.cnc_channel_r].nHliChannelIdx]^.channel_mc_control.mode_and_state.state_r.state = HLI_IMCM_PROCESS_RESETTING THEN
		stStatus.nCNCErrorID := 0;
		CNCSystem.LogAxisNo[gpAx[nHliIdx]^.head.log_ax_nr_r].nCNCErrorID := 0;
	ELSE
		stStatus.nCNCErrorID := CNCSystem.LogAxisNo[gpAx[nHliIdx]^.head.log_ax_nr_r].nCNCErrorID;	
	END_IF
END_IF
END_ACTION

END_FUNCTION_BLOCK

// CNC/3 Control/HLI3_SetAxisReferenceCam
FUNCTION HLI3_SetAxisReferenceCam : BOOL
VAR_INPUT
	nHliAxisIdx: INT;
	bReferenceCam: BOOL;
END_VAR
VAR
	/// Index of axis specific HLI area 
	nHliAxIfcIdx: INT;
END_VAR

(* ========================================================= *)
(*    FUN: HLI_SetAxisReferenceCam                           *)
(* --------------------------------------------------------- *)
(*   Desc:                                                   *)
(* Author: MK,MiB                                            *)
(*   Date: 30.11.2012                                        *)
(*   Rev.: 1.1                                               *)
(* ========================================================= *)


IF NOT HLI3_CheckAxisValid(nHliAxisIdx := nHliAxisIdx) THEN
	HLI3_SetAxisReferenceCam := FALSE;
	RETURN;
END_IF

(* set reference cam *)
gpAx[nHliAxisIdx]^.lr_mc_control.reference_cam.enable_w  := TRUE;
gpAx[nHliAxisIdx]^.lr_mc_control.reference_cam.command_w := bReferenceCam;

HLI3_SetAxisReferenceCam := TRUE;

END_FUNCTION

// CNC/3 Control/HLI3_SetAxisRelease
FUNCTION_BLOCK HLI3_SetAxisRelease
VAR_INPUT
	bEnable: BOOL;
	nHliAxisIdx: INT;
END_VAR
VAR_OUTPUT
	bAxisIsReady: BOOL;
	bAxisIsEnabled: BOOL;
	bAxisHasError: BOOL;
	nDriveType: UDINT;
	bError: BOOL;
	nErrorId: UDINT;
	nErrorState: UINT;
END_VAR
VAR
	bReadyForPowerOn: BOOL;
	bReadyForControlLoopOn: BOOL;
	nHliAxisIdxOld: INT;
	nState: UINT;
	nStateOld: UINT;
	tActiveTimeOut: TIME := TIME#5s0ms;
	wDriveState: WORD;
	fbTonTimeOut: TON;
END_VAR
VAR CONSTANT
	ERR_INVALID_AXIS_IDX: UDINT := 10000;
	ERR_UNSUPPORTED_DRIVE: UDINT := 10001;
	ERR_TIME_OUT: UDINT := 10002;
END_VAR

(****************************************************************************************)
(* POU:		HLI3_SetAxisRelease                      									*)
(* Type:	Function block																*)
(* Author: 	HR																			*)
(* Date: 	14/01/10																	*)
(* Rev.: 	1.0																			*)
(* ------------------------------------------------------------------------------------ *)
(* Author: 	TV																			*)
(* Date: 	14/04/11																	*)
(* Rev.: 	1.1																			*)
(* 			Implementation for terminal drives											*)
(* ------------------------------------------------------------------------------------ *)
(* Author: 	HR																			*)
(* Date: 	14/08/27																	*)
(* Rev.: 	1.2																			*)
(* 			Fixed terminal drive issue --> According to the ISG docs terminal drives	*)
(*			are supported by means of the torque permission control unit only! There-	*)
(*			fore this has to be switched by the 'bEnable' input. Tested with EL7041		*)
(* ------------------------------------------------------------------------------------ *)
(* Author: 	MiB																			*)
(* Date: 	16/04/06																	*)
(* Rev.: 	1.2																			*)
(* 			Enable follow up only for non simulation axis								*)
(* ------------------------------------------------------------------------------------ *)		
(* Desc:	Sets axes release and follow up mode using the axis specific control units 	*)
(*			'.lr_mc_control.torque_permission', 'lr_mc_control.release_feedhold',		*)
(*			'lr_mc_control.drive_on' and 'lr_mc_control.follow_up' depending on the 	*)
(*			subsequent drive type (e.g. Sercos,...). The following drive type are 		*)
(*			supported:																	*)
(*				+ Sercos and SoE														*)
(*				+ CanOpen and CoE (according to CiA402 drive profile)					*)
(*				+ Simulation drives														*)
(*																						*)
(*			This function block may raise the following error numbers					*)
(*				+ 10000	--> Invalid 'nHliAxisIdx'										*)
(*				+ 10001 --> Unsupported drive type										*)
(*				+ 10002 --> Time out while setting axis release							*)
(*																						*)
(*			IMPORTANT: This function block does not implement any state specific en- or	*)
(*			disabling of the drive. It simply tries to enable the subsequent axis as	*)
(*			long as input variable 'bEnable' is TRUE. That means it won´t disable the 	*)
(*			drive in case of any errors or loss prerequisited operation conditions (e.g.*)
(*			power supply). It is assumed that the drive will handle those situations	*)
(*			internally!																	*)
(*				  																		*)
(* 			Tested with following drives:												*)
(*																						*)
(*			VENDOR				MAKE					FW-VERSION			COM-SYS 	*)
(* 			------				----					----------			-------		*)
(* 			Beckhoff			AX5xxx					2.03 (B26)			SoE			*)
(* 			Beckhoff			EL7201					03					CoE			*)
(*			Beckhoff			EL7041					10					Terminal	*)	
(* 			ELMO				Gold					01.01.07.12			CoE			*)
(****************************************************************************************)

(****************************************************************************************)
(*									Check axis index									*)
(****************************************************************************************)
IF NOT HLI3_CheckAxisValid(nHliAxisIdx) THEN
	bError		:= TRUE;
	nErrorId	:= ERR_INVALID_AXIS_IDX;
	RETURN;
END_IF

(****************************************************************************************)
(*										Clear errors									*)
(****************************************************************************************)
IF bError THEN
	CASE nErrorId OF
	 (* -------------------------------------------------------------------------------	*)
	 ERR_INVALID_AXIS_IDX:
	 	(* Reset invalid HLI axis index error as soon as this line has been hit!		*)
		AC_ClearError();
		
	(* -------------------------------------------------------------------------------	*)
	 ERR_UNSUPPORTED_DRIVE:
		(* Reset unsupported drive type error in case the HLI axis index has been 		*)
		(* changed!																		*)
		IF (nHliAxisIdx <> nHliAxisIdxOld) THEN
			nHliAxisIdxOld	:= nHliAxisIdx;
			AC_ClearError();
		END_IF
 
	(* -------------------------------------------------------------------------------	*) 
	 ERR_TIME_OUT:
 		(* Will be resetted individually by each drive type specific action!			*)
	END_CASE
END_IF

(****************************************************************************************)
(*								Switch follow up mode 									*)
(****************************************************************************************)
IF gpAx[nHliAxisIdx]^.lr_state.drive_type_r = 4 THEN   (* type == 4 -> simulation axis -> don't enable follow up mode *)
	gpAx[nHliAxisIdx]^.lr_mc_control.follow_up.command_w := FALSE;
ELSE
	gpAx[nHliAxisIdx]^.lr_mc_control.follow_up.command_w := NOT bEnable;
END_IF

(****************************************************************************************)
(*						Copy axis state information to local variables					*)
(****************************************************************************************)
wDriveState				:= gpAx[nHliAxisIdx]^.lr_state.native_drive_state_r;
nDriveType				:= gpAx[nHliAxisIdx]^.lr_state.drive_type_r;
bAxisHasError			:= gpAx[nHliAxisIdx]^.lr_state.error_r;
bReadyForPowerOn		:= gpAx[nHliAxisIdx]^.lr_state.ready_for_power_on_r;
bReadyForControlLoopOn	:= gpAx[nHliAxisIdx]^.lr_state.ready_for_control_loop_on_r;

(****************************************************************************************)
(*							 Constant timeout implementation							*)
(****************************************************************************************)
IF (nStateOld <> nState) THEN
	nStateOld	:= nState;
	fbTonTimeOut(IN := FALSE);
END_IF

fbTonTimeOut
	(IN := TRUE,
	 PT := tActiveTimeOut
	);

(****************************************************************************************)
(*								Drive type specific axis release						*)
(****************************************************************************************)
CASE nDriveType OF
	HLI_DRIVE_CANOPEN	: AC_CanOpenDrive();
	HLI_DRIVE_SERCOS	: AC_SercosDrive();
	HLI_DRIVE_SIMU		: AC_SercosDrive();
	HLI_DRIVE_TERMINAL  : AC_TerminalDrive();
ELSE
	bError				:= TRUE;
	nErrorId			:= ERR_UNSUPPORTED_DRIVE;
END_CASE

ACTION AC_CanOpenDrive:
(****************************************************************************************)
(*										Status data										*)
(****************************************************************************************)
(* Ready state is signalled if the drive´s state is unequal to 'Not ready to switch on'	*)
bAxisIsReady	:= bReadyForControlLoopOn; 
 
(* Enabled state is derived from state 'Operation enabled' (information provided via	*)
(* HLI) and from status word bit no. 01 (switched on)!									*)
bAxisIsEnabled	:= bReadyForControlLoopOn AND bReadyForPowerOn AND wDriveState.1;

(****************************************************************************************)
(*						Command data (CanOpen requires a state machine)					*)
(****************************************************************************************)
(* Switch back to initial state in case the user want´s to disable the drive or an axis	*)
(* error occured, which requires a new srun of the sequence!							*)
IF NOT bEnable OR wDriveState.3 THEN
	nState				:= 0;
END_IF

CASE nState OF
 (* -----------------------------------------------------------------------------------	*)
 0: (* INIT *)
 	gpAx[nHliAxisIdx]^.lr_mc_control.torque_permission.command_w	:= FALSE;
 	gpAx[nHliAxisIdx]^.lr_mc_control.release_feedhold.command_w		:= FALSE;
	
	(* Start sequence in case the user wants to enable the drive and there is no error.	*)
 	IF bEnable AND NOT wDriveState.3 AND bAxisIsReady THEN
		(* Set time out once! *)
		tActiveTimeOut	:= T#2S;	
	
		// Switch on disabled???
		IF wDriveState.6 THEN
			nState		:= 10;
		//Ready to switch on???
		ELSIF wDriveState.0 THEN
			nState		:= 20;
		//Switched on???
		ELSIF wDriveState.1 THEN
			nState		:= 30;
		//Operation enabled???
		ELSIF wDriveState.2 THEN
			nState		:= 40;
		END_IF
	END_IF
	
 (* -----------------------------------------------------------------------------------	*)
 10: (* DRIVE IN 'Switch on disabled' STATE *)
 	gpAx[nHliAxisIdx]^.lr_mc_control.drive_on.command_w				:= TRUE;
 
	IF wDriveState.0 THEN
		nState			:= 20; 
	ELSIF fbTonTimeOut.Q THEN
		bError			:= TRUE;
		nErrorId		:= ERR_TIME_OUT;
		nErrorState		:= nState;
		nState			:= 0;
	END_IF
	
(* -----------------------------------------------------------------------------------	*)
 20: (* DRIVE IN 'Ready to switch on' STATE *)
 	gpAx[nHliAxisIdx]^.lr_mc_control.torque_permission.command_w	:= TRUE;
	
	IF wDriveState.1 THEN
		nState			:= 30; 
	ELSIF fbTonTimeOut.Q THEN
		bError			:= TRUE;
		nErrorId		:= ERR_TIME_OUT;
		nErrorState		:= nState;
		nState			:= 0;
	END_IF
	
 (* -----------------------------------------------------------------------------------	*)
 30: (* DRIVE IN 'Switched on' STATE *)
 	gpAx[nHliAxisIdx]^.lr_mc_control.release_feedhold.command_w		:= TRUE;
	
	IF wDriveState.2 THEN
		nState			:= 40; 
	ELSIF fbTonTimeOut.Q THEN
		bError			:= TRUE;
		nErrorId		:= ERR_TIME_OUT;
		nErrorState		:= nState;
		nState			:= 0;
	END_IF
	
 (* -----------------------------------------------------------------------------------	*)
 40: (* DRIVE IN 'Operation enabled' STATE *)
	AC_ClearError();
	
END_CASE
END_ACTION

ACTION AC_ClearError:
THIS^.bError		:= FALSE;
THIS^.nErrorId		:= 0;
THIS^.nErrorState	:= 0;
END_ACTION

ACTION AC_SercosDrive:
(****************************************************************************************)
(*										Status data										*)
(****************************************************************************************)
(* Ready state is derived from status word bit 15!										*)
bAxisIsReady	:= bReadyForControlLoopOn; 
 
(* Enabled state is derived from status word bits 14 and 15. IMPORTANT: In order to 	*)
(* take status word bit 03 into account  - which represents the time needed for 		*)
(* releasing the brake - axis specific parameter 'antr.sercos.evaluate_drive_follows_	*)
(* cmd' has to be set!!!																*) 
bAxisIsEnabled	:= bReadyForControlLoopOn AND bReadyForPowerOn;
 
(****************************************************************************************)
(*										Command data									*)
(****************************************************************************************)
(* ControlBit no. 14 is set statically in order to provide torque supported stopping of	*)
(* in case someone disables the axis during movement!									*) 
gpAx[nHliAxisIdx]^.lr_mc_control.torque_permission.command_w	:= TRUE;

(* Only control bits 13 and 15 are being (re-)set in order to achieve axis enabling!	*)
gpAx[nHliAxisIdx]^.lr_mc_control.release_feedhold.command_w		:= bEnable;
gpAx[nHliAxisIdx]^.lr_mc_control.drive_on.command_w				:= bEnable;
END_ACTION

ACTION AC_TerminalDrive:
(****************************************************************************************)
(*										Status data										*)
(****************************************************************************************)
(* Since there is no feedback available on the HLI axis enabled state wiöö be emulated!	*)
bAxisIsEnabled	:= bEnable;
bAxisIsReady	:= FALSE;
 
(****************************************************************************************)
(*										Command data									*)
(****************************************************************************************)
(* Terminal drives are supported by the torque permission control unit only!			*)
gpAx[nHliAxisIdx]^.lr_mc_control.torque_permission.command_w	:= bEnable;
gpAx[nHliAxisIdx]^.lr_mc_control.release_feedhold.command_w		:= FALSE;
gpAx[nHliAxisIdx]^.lr_mc_control.drive_on.command_w				:= FALSE;
END_ACTION

END_FUNCTION_BLOCK

// CNC/3 Control/HLI3_SetAxisReferenceOffset
FUNCTION_BLOCK HLI3_SetAxisReferenceOffset
VAR_INPUT
	Execute: BOOL;
	nHliAxisIdx: INT;
	nOffset:	LREAL;  (* Offset in mm *)
END_VAR
VAR_OUTPUT
	Busy  : BOOL;
	Done: BOOL;
	Error : BOOL;
	ErrorId : INT;
END_VAR
VAR
	nState : int;
	trigStart: R_TRIG;
END_VAR

(* ========================================================= *)
(*    FUN: HLI3_SetAxisReferenceOffset                      *)
(* --------------------------------------------------------- *)
(*   
    Desc: 
	Set reference offset position of an axis.
 
	To use this FB to set the offset for absolute encoder axis the following axis parameter settings should be done:
	
	kenngr.abs_pos_gueltig	0			( P-AXIS-00014 : Identification code for absolute path measurement system
	kenngr.set_refpos_mode	PLC_OFFSET  ( P-AXIS-00278 : Modes for setting the homing position (ABSOLUT / OFFSET /  PLC / PLC_OFFSET)
	
	While commanding the axis must not be involved in active interpolation or active manual mode!
	
	Errors:
	1 : nHliAxisIdx is invalid
*)
(*                                               
   Author: MiB                                               
   Date: 13.07.2017                                        
   Rev.: 1.0                                               
 =========================================================*) 
 
 trigStart(clk := Execute);
 IF trigStart.Q THEN  // start on flank of Execute
		 nState := 10;    
		 Done := FALSE;
		 Error := FALSE;
		 ErrorId := 0;
		 Busy := TRUE;
		gpAx[nHliAxisIdx]^.lr_mc_control.set_reference_position.command_w := FALSE;	 
		gpAx[nHliAxisIdx]^.lr_mc_control.clear_reference_position.command_w := FALSE;
 END_IF
 
 CASE nState OF
	 0: (* Idle *)
	 	Done := TRUE;
		Busy := FALSE;
	10: (* check Axis id valid *)
		IF NOT HLI3_CheckAxisValid(nHliAxisIdx := nHliAxisIdx) THEN	
			nState :=-1;
			Done := TRUE;
			Busy := FALSE;
			Error := TRUE;
			ErrorId := 1;		
		ELSE
			nState := nState + 10;		
		END_IF		
	20: (* Start *)
		(* set reference position *)
		gpAx[nHliAxisIdx]^.lr_mc_control.clear_reference_position.enable_w := TRUE;
		gpAx[nHliAxisIdx]^.lr_mc_control.clear_reference_position.command_w := TRUE;
		IF gpAx[nHliAxisIdx]^.lr_mc_control.clear_reference_position.state_r THEN
			gpAx[nHliAxisIdx]^.lr_mc_control.clear_reference_position.command_w := FALSE;
			nState := nState + 10;
		END_IF

	30: (* transfer new offset value *)
		gpAx[nHliAxisIdx]^.lr_mc_control.refpos_position.command_w := LREAL_TO_DINT(nOffset *10000.0);
		IF (gpAx[nHliAxisIdx]^.lr_mc_control.refpos_position.state_r = LREAL_TO_DINT(nOffset * 10000.0) ) THEN
			gpAx[nHliAxisIdx]^.lr_mc_control.set_reference_position.command_w := TRUE;
			nState := nState + 10;		
		END_IF
	40: (* tigger "write offset" *)
		
		IF (gpAx[nHliAxisIdx]^.lr_mc_control.set_reference_position.state_r) THEN
			gpAx[nHliAxisIdx]^.lr_mc_control.set_reference_position.command_w := FALSE;
			nState := 0;
		END_IF
	
	
 END_CASE

END_FUNCTION_BLOCK

// CNC/3 Control/HLI3_ClearReferencePosition
FUNCTION HLI3_ClearReferencePosition : BOOL
VAR_INPUT
	bExecute: BOOL;
	nHliAxisIdx: INT;
END_VAR

(* ========================================================= *)
(*    FUN: HLI3_ClearReferencePosition                       *)
(* --------------------------------------------------------- *)
(*   Desc:                                                   *)
(* 	 Author: TV                                              *)
(*   Date: 17.06.2015                                        *)
(*   Rev.: 1.0                                               *)
(* ========================================================= *)
HLI3_ClearReferencePosition := FALSE;

IF NOT HLI3_CheckAxisValid(nHliAxisIdx := nHliAxisIdx) THEN	
	RETURN;
END_IF

(* set reference position *)
gpAx[nHliAxisIdx]^.lr_mc_control.clear_reference_position.enable_w := TRUE;
gpAx[nHliAxisIdx]^.lr_mc_control.clear_reference_position.command_w := bExecute;
HLI3_ClearReferencePosition := TRUE;

END_FUNCTION

// CNC/3 Control/HLI3_SetProbingSignal
FUNCTION HLI3_SetProbingSignal : BOOL
VAR_INPUT
	nHliAxisIdx: INT;
	bProbingSignal: BOOL;
END_VAR


IF NOT HLI3_CheckAxisValid(nHliAxisIdx := nHliAxisIdx) THEN	
	HLI3_SetProbingSignal := FALSE;
	RETURN;
END_IF


gpAx[nHliAxisIdx]^.lr_mc_control.probing_signal.enable_w  := TRUE;
gpAx[nHliAxisIdx]^.lr_mc_control.probing_signal.command_w := bProbingSignal;
HLI3_SetProbingSignal := TRUE;

END_FUNCTION

// CNC/12 CNC_Axis/FB_ReadSWLimitSwitches
//*********************************************************************************************************
///NAME.......................:		FB_ReadSWLimitSwitches
///DATUM....................:		03.01.2018
///AUTOR....................:		Thomas Voß
///VERSION................:			1.1
///
///Description.: 	Read Software Limit Switches					
///**********************************************************************************************************

FUNCTION_BLOCK FB_ReadSWLimitSwitches
VAR_INPUT	
	nLogAxisNo		: UINT;		
	bExecute		: BOOL;
END_VAR
VAR_OUTPUT
	bError : BOOL;
	bBusy: BOOL;
	fSWLimitNeg		: LREAL;	(* Unit mm *)
	fSWLimitPos		: LREAL;	(* Unit mm *)
END_VAR
VAR
		fbOnTrigger		:  	R_TRIG;
		FbAdsRead		: 	ADSREAD;
		Step 			: 	UDINT;
		TimeOut 		: 	TON;	
		nSWLimitNeg 	: 	DINT;
		nSWLimitPos  	: 	DINT;
END_VAR

fbOnTrigger(CLK:= bExecute);


IF fbOnTrigger.Q THEN
	Step 	:= 10;	
	bError	:= 0;
	bBusy 	:= TRUE;
	FbAdsRead(READ := FALSE);
	
	fSWLimitNeg		:= 0;
	fSWLimitPos		:= 0;
	nSWLimitNeg 	:= 0;
	nSWLimitPos  	:= 0;
END_IF

CASE Step OF
0:
	bBusy 	:= FALSE;
	
10: (* Read negative Limit Switch *)

	IF nLogAxisNo < 1 OR  nLogAxisNo > MAX_SYS_LOG_AXIS_INDEX THEN
		Step := 999;
	ELSIF CNCSystem.LogAxisNo[nLogAxisNo].nHliAxisIdx = -1 THEN
		Step := 999;
	ELSE
		TimeOut(IN:=FALSE);
		FbAdsRead(	NETID:= '',							(* local *)
					PORT:= 553,							(* Port number of Task COM, all ADS-Requests to the NC-kernel  *)                          
					IDXGRP:=16#00020200+nLogAxisNo,    	(*  *)
					IDXOFFS:= 16#26,
					LEN:=SIZEOF(nSWLimitNeg),		(* number of bytes that shall be read                          *)
					DESTADDR:= ADR(nSWLimitNeg),  	(* memory for the read value, must be provided by the user     *)
					READ:=TRUE,							(* a rising edge on this input starts the read request         *)
					TMOUT:= T#1S);       				(* maximum time for read request                               *)
	
			Step := Step+10;
	END_IF

20:
		TimeOut(IN:=TRUE, PT:=T#2S);
		FbAdsRead();
		IF NOT FbAdsRead.Busy THEN
			IF NOT FbAdsRead.ERR THEN
				FbAdsRead(READ := FALSE);				
				fSWLimitNeg	 := DINT_TO_LREAL(nSWLimitNeg) / 10000.0; 				
				Step := Step+10;
			ELSE
				FbAdsRead(READ := FALSE);				
				Step := 999;
			END_IF
		END_IF

		(* error timeout *)
		IF TimeOut.Q THEN			
			Step   	:= 999;
		END_IF

30: (* Read positive Limit Switch *)
	TimeOut(IN:=FALSE);
	FbAdsRead(	NETID:= '',							(* local *)
				PORT:= 553,							(* Port number of Task COM, all ADS-Requests to the NC-kernel  *)
				IDXGRP:=16#00020200+nLogAxisNo,     (*  *)
				IDXOFFS:= 16#25,
				LEN:=SIZEOF(nSWLimitPos),		(* number of bytes that shall be read                          *)
				DESTADDR:= ADR(nSWLimitPos),  	(* memory for the read value, must be provided by the user     *)
				READ:=TRUE,							(* a rising edge on this input starts the read request         *)
				TMOUT:= T#1S);       				(* maximum time for read request                               *)
				
				Step := Step+10;

40:	TimeOut(IN:=TRUE, PT:=T#2S);
		FbAdsRead();
		IF NOT FbAdsRead.Busy THEN
			IF NOT FbAdsRead.ERR THEN
				FbAdsRead(READ := FALSE);
				fSWLimitPos	 := DINT_TO_LREAL(nSWLimitPos) / 10000.0;
				Step := 0;
			ELSE
				FbAdsRead(READ := FALSE);				
				Step := 999;
			END_IF
		END_IF
		
		(* error timeout *)
		IF TimeOut.Q THEN			
			Step   	:= 999;
		END_IF

		
999:	(* Error *)
		bError := TRUE;
		Step := 0;	
	
END_CASE

END_FUNCTION_BLOCK

// CNC/12 CNC_Axis/HLI3_CNCAxis
FUNCTION_BLOCK HLI3_CNCAxis EXTENDS HLI3_CNCAxisBase
VAR_INPUT
	nHliAxisIdx : INT := -1;
END_VAR
VAR_OUTPUT
END_VAR
VAR
END_VAR

(* ========================================================= *)
(*     FB: HLI3_CNCAxis                                  	 *)
(* --------------------------------------------------------- *)
(*   Desc:  CNC Axis Control							   	 *)
(*   Author: TV				                                 *)
(*   Date: 2018.01.25                                        *)
(*   Rev.: 1.0                                               *)
(* ==========================================================*)

SUPER^(nHliIdx := nHliAxisIdx);

END_FUNCTION_BLOCK

// CNC/2 OperationMode/ModeManual/HLI3_LogicalAxisInManualMode
FUNCTION HLI3_LogicalAxisInManualMode : ARRAY[0..HLI_KEY_MAXIDX] OF UINT
VAR_INPUT
	nChan: INT;
END_VAR
VAR
	i: INT;
	n: INT;
END_VAR

(* 		  If no axis is in manual mode it returns 0           		*)
(* Author: MiB/TV                                         			*)
(*   Date: 16.07.2007                                         		*)
(*   Last: 05.04.2016                                        		*)
(*   Rev.: 1.1                                                 		*)
(* ================================================================= *)

IF (NOT HLI3_CheckChannelValid(nChannel := nChan)) THEN
	RETURN;
END_IF

n:= 0;
FOR i := 0 TO HLI_CH_AX_MAXIDX DO
  	IF (gpCh[nChan]^.bahn_state.coord_r[i].hb_display_r.state <> 0) THEN
		HLI3_LogicalAxisInManualMode[n] := gpCh[nChan]^.bahn_state.coord_r[i].log_achs_nr_r;
		IF n < HLI_KEY_MAXIDX THEN
			n := n+1;
		END_IF
	END_IF
END_FOR

END_FUNCTION

// CNC/2 OperationMode/ModeManual/HLI3_ManualActivation
FUNCTION_BLOCK HLI3_ManualActivation
VAR_INPUT
	bExecute: BOOL;
	/// Number of channel 
	nChan: INT;
	eManualType: E_CNC_ManualType;
	/// Increments -> 0 activates Tip mode 
	Inc: UDINT;
	/// Aufloesung des Achsverfahrwegs bei einer Handradumdrehung Einheit: 0.1um / Handradumdrehung
	nHBA_Res: DINT;
	Speed: UDINT;
	/// axis nr 
	nLogAxisNr: UINT;
	nInputParameterIdx: INT;
END_VAR
VAR_OUTPUT
	bError: BOOL;
	bBusy: BOOL;
END_VAR
VAR_IN_OUT
	stManualModeControlElements: ST_ManualModeControlElements;
	stManualModeControlElementState: ST_ManualModeControlElementState;
END_VAR
VAR
	fbRtrigExec: R_TRIG;
	nState: INT;
	pActivation: POINTER TO MC_CONTROL_HB_ACTIVATION_UNIT;
	pJogParameter: POINTER TO MC_CONTROL_HB_JOG_PARAM_UNIT;
	pTipParameter: POINTER TO MC_CONTROL_HB_TIP_PARAM_UNIT;
	pHBHRParameter: POINTER TO MC_CONTROL_HB_HR_PARAM_UNIT;
	j: INT;
	bFreeControlElementFound: BOOL;
END_VAR

(* ========================================================= *)
(*    FUN: HLI_ManualActivation                       		 *)
(* --------------------------------------------------------- *)
(*   Desc:                                                   *)
(*   Author: CL TV MiB                                       *)
(*   Date: 18.11.2005                                        *)
(*   Last: 06.06.2017                                       *)
(*   Rev.: 6.2                                              *)
(* ========================================================= *)

IF NOT HLI3_CheckChannelValid(nChannel := nChan) OR nLogAxisNr = 0 THEN
	RETURN;
END_IF


fbRtrigExec(clk := bExecute);
IF fbRtrigExec.Q THEN
	bBusy := TRUE;
	bError := FALSE;
	nState := 10;
END_IF

CASE nState OF

	0: (* IDLE *)
		bBusy := FALSE;

	10:
		CASE eManualType OF
			E_CNC_ManualType.NoManualMode: 
				nState := 100;

			E_CNC_ManualType.Handwheel:
				nState := 30;

			E_CNC_ManualType.TippMode:
				nState := 40;

			E_CNC_ManualType.JogMode:
				nState := 50;

			E_CNC_ManualType.JoystickMode:
				nState := 40;

			E_CNC_ManualType.DigitalJoystick: 
				nState := 40;

		END_CASE

	30:(* Setze Handrad Parameter *)
		pHBHRParameter := ADR(gpCh[nChan]^.hb_mc_control.hr_parameter);
		IF NOT pHBHRParameter^.command_semaphor_rw THEN
			pHBHRParameter^.enable_w := TRUE;
			pHBHRParameter^.command_w.resolution  := nHBA_Res;
			pHBHRParameter^.command_w.log_achs_nr := nLogAxisNr;
			pHBHRParameter^.command_semaphor_rw := TRUE;
			nState := 100;
		END_IF

	40: (* Setze Parameter für den Tippbetrieb *)
		pTipParameter := ADR(gpCh[nChan]^.hb_mc_control.tip_parameter);
		IF NOT pTipParameter^.command_semaphor_rw THEN
			pTipParameter^.enable_w := TRUE;
			pTipParameter^.command_w.log_achs_nr := nLogAxisNr;
			pTipParameter^.command_w.speed       := Speed;
			pTipParameter^.command_semaphor_rw := TRUE;
			nState := 100;
		END_IF

	50: (* Setze Parameter für den Jogbetrieb *)
		pJogParameter := ADR(gpCh[nChan]^.hb_mc_control.jog_parameter);
		IF NOT pJogParameter^.command_semaphor_rw THEN
			pJogParameter^.enable_w := TRUE;
			pJogParameter^.command_w.log_achs_nr := nLogAxisNr;
			pJogParameter^.command_w.distance    := Inc;
			pJogParameter^.command_w.speed       := Speed;
			pJogParameter^.command_semaphor_rw := TRUE;
			nState := 100;
		END_IF		
		
	100: 	(* Aktivierung der Bedienelementen für den Handbetrieb  *)
		pActivation := ADR(gpCh[nChan]^.hb_mc_control.activation);						
		IF 	NOT gpCh[nChan]^.hb_mc_control.activation.command_semaphor_rw AND 
			NOT gpCh[nChan]^.hb_mc_control.tip_parameter.command_semaphor_rw AND 
		   	NOT gpCh[nChan]^.hb_mc_control.jog_parameter.command_semaphor_rw AND 
		   	NOT gpCh[nChan]^.hb_mc_control.hr_parameter.command_semaphor_rw
		THEN 
			bFreeControlElementFound := FALSE;

			IF 	eManualType <> E_CNC_ManualType.Handwheel THEN 	
				FOR j := 0 TO HLI_KEY_MAXIDX DO
					IF stManualModeControlElementState.stKeyUnit[j].nLogAxisId = 0 THEN
							stManualModeControlElementState.stKeyUnit[j].nLogAxisId := nLogAxisNr;
							stManualModeControlElementState.stKeyUnit[j].nChan := nChan;
							stManualModeControlElementState.stKeyUnit[j].nInputParameterIdx := nInputParameterIdx;
							bFreeControlElementFound := TRUE;
						EXIT;
					END_IF 
				END_FOR
			ELSE
				FOR j := 0 TO HLI_HW_MAXIDX DO
					IF stManualModeControlElementState.stHWUnit[j].nLogAxisId = 0 THEN
							stManualModeControlElementState.stHWUnit[j].nLogAxisId := nLogAxisNr;
							stManualModeControlElementState.stHWUnit[j].nChan := nChan;
							stManualModeControlElementState.stHWUnit[j].nInputParameterIdx := nInputParameterIdx;
							bFreeControlElementFound := TRUE;
						EXIT;
					END_IF 
				END_FOR
			END_IF
							
			IF bFreeControlElementFound THEN
				pActivation^.enable_w := TRUE;
				pActivation^.command_w.log_achs_nr := nLogAxisNr;
				pActivation^.command_w.control_element := INT_TO_UINT(j+1);
		
		
				CASE eManualType OF
					E_CNC_ManualType.NoManualMode: 
						pActivation^.command_w.operation_mode := 0; 	(* 0 - No OP_Mode *)
		
					E_CNC_ManualType.Handwheel: 
						gpCh[0]^.hb_mc_control.handwheel_incs[j].command_w := stManualModeControlElements.nHandwheelInc[stManualModeControlElementState.stHWUnit[j].nInputParameterIdx];
						pActivation^.command_w.operation_mode := 1; 	(* 1 - Handwheel *)
		
					E_CNC_ManualType.TippMode: 
						pActivation^.command_w.operation_mode := 2; 	(* 2 - Tip Mode continous *)
		
					E_CNC_ManualType.JogMode: 
						pActivation^.command_w.operation_mode := 3; 	(* 3 - Jog Mode (incremental *)
		
					E_CNC_ManualType.JoystickMode: 
						pActivation^.command_w.operation_mode := 2; 	(* 2 - Tip Mode continous, auch für Analog Joystick *)
		
					E_CNC_ManualType.DigitalJoystick: 
						pActivation^.command_w.operation_mode := 2; 	(* 2 - Tip Mode continous, auch für Digital Joystick *)
		
				END_CASE
			
				pActivation^.command_semaphor_rw := TRUE;
				nState := 110;
			ELSE
				bError := TRUE;
				nState := 0;
			END_IF
		END_IF		

	110:	
		IF  NOT gpCh[nChan]^.hb_mc_control.activation.command_semaphor_rw  THEN 		
			nState := 0;
		END_IF
			
END_CASE

END_FUNCTION_BLOCK

// CNC/2 OperationMode/ModeManual/HLI3_ManualExecution
FUNCTION_BLOCK HLI3_ManualExecution
VAR_INPUT
	nChan: INT;
	/// number of the HB_KeyControlUnit 
	nKeyControlUnit: INT;
	/// static signal 
	bKeyPos: BOOL;
	/// static signal 
	bKeyNeg: BOOL;
END_VAR
VAR
	Cmd_Dir: E_HLI_MM_KEYDirection;
	Act_Dir: E_HLI_MM_KEYDirection;
END_VAR

(* ========================================================= *)
(*    FUN: HLI_ManualExecution                    		 		 *)
(* --------------------------------------------------------- *)
(*   Desc:                                                   *)
(*   Author: CL / TV                                         *)
(*   Date: 24.07.2015                                       *)
(*   Rev.: 6.0                                               *)
(* ========================================================= *)

(* flank detection second axis*)
gpCh[nChan]^.hb_mc_control.key[nKeyControlUnit].enable_w := TRUE;

IF (NOT bKeyPos AND NOT bKeyNeg) OR (bKeyPos AND Act_Dir = KEY_DIR_NEGATIVE) OR (bKeyNeg AND Act_Dir = KEY_DIR_POSITIVE) THEN
	Cmd_Dir := KEY_DIR_NOT_PRESSED;
	IF NOT gpCh[nChan]^.hb_mc_control.key[nKeyControlUnit].command_semaphor_rw AND Cmd_dir <> Act_Dir THEN
		gpCh[nChan]^.hb_mc_control.key[nKeyControlUnit].command_w.log_key_nr := DINT_TO_UINT(nKeyControlUnit)+1;
		gpCh[nChan]^.hb_mc_control.key[nKeyControlUnit].command_w.direction := KEY_DIR_NOT_PRESSED;
		gpCh[nChan]^.hb_mc_control.key[nKeyControlUnit].command_semaphor_rw := TRUE;
		Act_Dir := KEY_DIR_NOT_PRESSED;
	END_IF	
END_IF


IF bKeyPos AND Act_Dir = KEY_DIR_NOT_PRESSED THEN
	Cmd_Dir := KEY_DIR_POSITIVE;
	IF NOT gpCh[nChan]^.hb_mc_control.key[nKeyControlUnit].command_semaphor_rw AND Cmd_dir <> Act_Dir THEN
		gpCh[nChan]^.hb_mc_control.key[nKeyControlUnit].command_w.log_key_nr := DINT_TO_UINT(nKeyControlUnit)+1;
		gpCh[nChan]^.hb_mc_control.key[nKeyControlUnit].command_w.direction := KEY_DIR_POSITIVE;
		gpCh[nChan]^.hb_mc_control.key[nKeyControlUnit].command_semaphor_rw := TRUE;
		Act_Dir := KEY_DIR_POSITIVE;
	END_IF	
END_IF

IF bKeyNeg AND Act_Dir = KEY_DIR_NOT_PRESSED  THEN
	Cmd_Dir := KEY_DIR_NEGATIVE;
	IF NOT gpCh[nChan]^.hb_mc_control.key[nKeyControlUnit].command_semaphor_rw AND Cmd_dir <> Act_Dir THEN
		gpCh[nChan]^.hb_mc_control.key[nKeyControlUnit].command_w.log_key_nr := DINT_TO_UINT(nKeyControlUnit)+1;
		gpCh[nChan]^.hb_mc_control.key[nKeyControlUnit].command_w.direction := KEY_DIR_NEGATIVE;
		gpCh[nChan]^.hb_mc_control.key[nKeyControlUnit].command_semaphor_rw := TRUE;
		Act_Dir := KEY_DIR_NEGATIVE;
	END_IF	
END_IF

END_FUNCTION_BLOCK

// CNC/2 OperationMode/ModeManual/HLI3_ManualExecutionRapidMode
FUNCTION_BLOCK HLI3_ManualExecutionRapidMode
VAR_INPUT
	nChan: INT;
	/// number of the HB_KeyControlUnit 
	nKeyControlUnit: INT;
	/// static signal 
	bExecute: BOOL;
END_VAR
VAR
	pRapidKey: POINTER TO MC_CONTROL_HB_RAPID_KEY_UNIT;
	TONTimeOut: TON;
	fbRtrigExec: R_TRIG;
	fbFtrigExec: F_TRIG;
END_VAR

(* ========================================================= *)
(*    FUN: HLI_ManualExecution                               *)
(* --------------------------------------------------------- *)
(*   Desc:                                                   *)
(*   Author: TV                                              *)
(*   Date: 24.07.2015                                        *)
(*   Rev.: 6.0                                               *)
(* ========================================================= *)


IF nKeyControlUnit < 0 OR nKeyControlUnit > HLI_KEY_MAXIDX THEN
	RETURN;
END_IF;

pRapidKey := ADR(gpCh[nChan]^.hb_mc_control.rapid_key);
pRapidKey^.enable_w := TRUE;

IF NOT pRapidKey^.command_semaphor_rw THEN
	fbRtrigExec(clk := bExecute);
	fbFtrigExec(clk := bExecute);
END_IF

IF fbRtrigExec.Q THEN
	pRapidKey^.command_w.key_pressed := 1;
	pRapidKey^.command_w.log_key_nr := INT_TO_UINT(nKeyControlUnit)+1;
	pRapidKey^.command_semaphor_rw := TRUE;
END_IF


IF fbFtrigExec.Q THEN
	pRapidKey^.command_w.key_pressed := 0;
	pRapidKey^.command_w.log_key_nr := INT_TO_UINT(nKeyControlUnit)+1;
	pRapidKey^.command_semaphor_rw := TRUE;
END_IF

END_FUNCTION_BLOCK

// CNC/2 OperationMode/ModeManual/HLI3_ManualModeHandler
FUNCTION_BLOCK HLI3_ManualModeHandler
VAR_INPUT
	stManualModeParameter: ST_ManualModeParameter;
	stManualModeControlElements: ST_ManualModeControlElements;
	bReset: BOOL;
END_VAR
VAR_OUTPUT
	bInManualMode: BOOL;
	arrAxisInG201: ARRAY[0..HLI_KEY_MAXIDX] OF UINT;
	bBusy: BOOL;
	bError: BOOL;
	nErrorId: INT;
END_VAR
VAR_IN_OUT
	stManualModeControlElementState : ST_ManualModeControlElementState;
	stCmdModesStates    			: ST_CNCCmdModesStates;
END_VAR
VAR
	nState: INT;
	pString: POINTER TO STRING;
	pUnit: POINTER TO MC_CONTROL_MCM_MODE_STATE_UNIT;
	pCommand: POINTER TO HLI_PROC_TRANS_TO_MODE_STATE;
	pKey: POINTER TO MC_CONTROL_HB_KEY_UNIT;
	pIncr: POINTER TO MC_CONTROL_HB_TIP_PARAM_UNIT;
	stManualModeParameterOld: ST_ManualModeParameter;
	incOld: UINT;
	nManualTypOld: UINT;
	i: INT;
	bManual: BOOL;
	/// FBs for manual mode 
	ManualActivation: HLI3_ManualActivation;
	ManualExecution: ARRAY[0..HLI_KEY_MAXIDX] OF HLI3_ManualExecution;
	ManualExecutionRapidMode: ARRAY[0..HLI_KEY_MAXIDX] OF HLI3_ManualExecutionRapidMode;
	ActChannelModeOld: UDINT;
	TON_TimeOut: TON;
	nChan: INT;
	j: INT;
	strInitParameterOld: STRING;
	bInJoystickMode: BOOL;
	nHliAxisIdx: INT;
	nControlUnit: INT;
	arrAxisInJoystickMode: ARRAY[0..HLI_KEY_MAXIDX] OF UINT;
	n: INT;
	bInit: BOOL;
	strInitParameter : STRING;	
	strZeroOffset : STRING;
END_VAR
VAR CONSTANT
	ErrID_1: INT := 1;
END_VAR

(* ========================================================= 	*)
(*     FB: HLI3_ManualModeHandler                           	*)
(* --------------------------------------------------------- 	*)
(*   Desc: Switch to Manual Mode and parametrize             	*)
(*   Author: MK / TV  /MiB                                      *)
(*   Date: 18.07.2002                                        	*)
(*   Last: 23.10.2017                                        	*)
(*   Rev.: 6.7	                                              	*)
(* ========================================================= 	*)

nChan := stManualModeParameter.stChannelParameter.nChanIdx;
IF (NOT HLI3_CheckChannelValid(nChannel := nChan) OR nChan = -1 )  THEN
	RETURN;
END_IF

IF NOT bInit THEN  
	gpCh[nChan]^.hb_mc_control.activation.enable_w := TRUE;
	FOR j := 0 TO HLI_HW_MAXIDX DO
		gpCh[nChan]^.hb_mc_control.handwheel_incs[j].enable_w  := TRUE;
	END_FOR
	bInit := TRUE;
END_IF	

IF 	CNCSystem.Channel[nChan].ActMode <> HLI_IMCM_MANUAL_MODE AND
	CNCSystem.Channel[nChan].ActMode <> HLI_IMCM_AUTOMATIC_MODE   AND
	CNCSystem.Channel[nChan].ActMode <> HLI_IMCM_MDI_MODE THEN
		strInitParameterOld := '';
		bBusy := FALSE;
		nState := 0;
	RETURN; (* A b b r u c h *)
ELSE
	bManual := TRUE;
END_IF

IF  CNCSystem.Channel[nChan].ActMode <> HLI_IMCM_MANUAL_MODE OR
	CNCSystem.Channel[nChan].ActState <> HLI_IMCM_PROCESS_ACTIVE THEN
	strInitParameterOld := '';
END_IF

(* Clear all request from the HMI *)
IF gpCh[nChan]^.hb_mc_control.key[0].request_semaphor_rw THEN
	gpCh[nChan]^.hb_mc_control.key[0].request_semaphor_rw := FALSE;
END_IF

IF gpCh[nChan]^.hb_mc_control.activation.request_semaphor_rw THEN
	gpCh[nChan]^.hb_mc_control.activation.request_semaphor_rw := FALSE;
END_IF

IF gpCh[nChan]^.hb_mc_control.tip_parameter.request_semaphor_rw THEN
	gpCh[nChan]^.hb_mc_control.tip_parameter.request_semaphor_rw := FALSE;
END_IF

IF gpCh[nChan]^.hb_mc_control.jog_parameter.request_semaphor_rw THEN
	gpCh[nChan]^.hb_mc_control.jog_parameter.request_semaphor_rw := FALSE;
END_IF

bBusy := TRUE;

IF bReset THEN		
	bError := FALSE;
	nErrorID := 0;
	bInManualMode := FALSE;
END_IF


IF stManualModeParameter.stChannelParameter.eManualType = E_CNC_ManualType.JoystickMode THEN

	bInJoystickMode := TRUE;
	
	arrAxisInJoystickMode := HLI3_LogicalAxisInManualMode(nCHan);
	
	PRG_AnalogJoystick(	nLogAxisNr:= stManualModeParameter.stAxisParameter.stControlUnit[0].nLogAxisNr,
								Analog_Value:= stManualModeControlElements.stControlJoystickValue[0],
								AnalogValueMin:= stManualModeParameter.stJoystickParameter.AnalogValueMin,
								AnalogValueMax:= stManualModeParameter.stJoystickParameter.AnalogValueMax,
								AnalogValueZeroDeadBand:= stManualModeParameter.stJoystickParameter.AnalogValueZeroDeadBand,
								bKeyPos:= stManualModeControlElements.stControlKeys[0].bKeyPos,
								bKeyNeg:= stManualModeControlElements.stControlKeys[0].bKeyNeg);

	PRG_AnalogJoystick(	nLogAxisNr:= stManualModeParameter.stAxisParameter.stControlUnit[1].nLogAxisNr,
								Analog_Value:= stManualModeControlElements.stControlJoystickValue[1],
								AnalogValueMin:= stManualModeParameter.stJoystickParameter.AnalogValueMin,
								AnalogValueMax:= stManualModeParameter.stJoystickParameter.AnalogValueMax,
								AnalogValueZeroDeadBand:= stManualModeParameter.stJoystickParameter.AnalogValueZeroDeadBand,
								bKeyPos:= stManualModeControlElements.stControlKeys[1].bKeyPos,
								bKeyNeg:= stManualModeControlElements.stControlKeys[1].bKeyNeg);

	PRG_AnalogJoystick(	nLogAxisNr:= stManualModeParameter.stAxisParameter.stControlUnit[2].nLogAxisNr,
								Analog_Value:= stManualModeControlElements.stControlJoystickValue[2],
								AnalogValueMin:= stManualModeParameter.stJoystickParameter.AnalogValueMin,
								AnalogValueMax:= stManualModeParameter.stJoystickParameter.AnalogValueMax,
								AnalogValueZeroDeadBand:= stManualModeParameter.stJoystickParameter.AnalogValueZeroDeadBand,
								bKeyPos:= stManualModeControlElements.stControlKeys[2].bKeyPos,
								bKeyNeg:= stManualModeControlElements.stControlKeys[2].bKeyNeg);

	PRG_AnalogJoystick(	nLogAxisNr:= stManualModeParameter.stAxisParameter.stControlUnit[3].nLogAxisNr,
								Analog_Value:= stManualModeControlElements.stControlJoystickValue[3],
								AnalogValueMin:= stManualModeParameter.stJoystickParameter.AnalogValueMin,
								AnalogValueMax:= stManualModeParameter.stJoystickParameter.AnalogValueMax,
								AnalogValueZeroDeadBand:= stManualModeParameter.stJoystickParameter.AnalogValueZeroDeadBand,
								bKeyPos:= stManualModeControlElements.stControlKeys[3].bKeyPos,
								bKeyNeg:= stManualModeControlElements.stControlKeys[3].bKeyNeg);

	PRG_AnalogJoystick(	nLogAxisNr:= stManualModeParameter.stAxisParameter.stControlUnit[4].nLogAxisNr,
								Analog_Value:= stManualModeControlElements.stControlJoystickValue[4],
								AnalogValueMin:= stManualModeParameter.stJoystickParameter.AnalogValueMin,
								AnalogValueMax:= stManualModeParameter.stJoystickParameter.AnalogValueMax,
								AnalogValueZeroDeadBand:= stManualModeParameter.stJoystickParameter.AnalogValueZeroDeadBand,
								bKeyPos:= stManualModeControlElements.stControlKeys[4].bKeyPos,
								bKeyNeg:= stManualModeControlElements.stControlKeys[4].bKeyNeg);

ELSE
	(* Achsoverride wieder auf 100 % setzen *)
	IF bInJoystickMode THEN 
		nHliAxisIdx := -1;
		FOR j := 0 TO UINT_TO_INT(SIZEOF(arrAxisInJoystickMode)) DO
			FOR i := 0 TO UDINT_TO_INT(gNrAx-1) DO
				IF (gpAX[i]^.head.log_ax_nr_r = arrAxisInJoystickMode[j]) THEN
					nHliAxisIdx := i;	
					IF (nHliAxisIdx <> -1) THEN 
						HLI3_SetAxisOverride(nHliAxisIdx := nHliAxisIdx, nOverride := 1000);
						nHliAxisIdx := -1;
						arrAxisInJoystickMode[j] := 0;
					END_IF								
				END_IF
			END_FOR			
		END_FOR
		bInJoystickMode := FALSE;
	END_IF
END_IF

(******** Parallelinterpolation mit G201 *************************************)
IF CNCSystem.Channel[nChan].ActMode = HLI_IMCM_AUTOMATIC_MODE OR CNCSystem.Channel[nChan].ActMode = HLI_IMCM_MDI_MODE THEN
	arrAxisInG201 := HLI3_LogicalAxisInManualMode(nCHan);
	FOR j := 0 TO HLI_KEY_MAXIDX DO
		stManualModeParameter.stAxisParameter.stControlUnit[j].nLogAxisNr := arrAxisInG201[j];
	END_FOR
ELSE
	FOR j := 0 TO HLI_KEY_MAXIDX DO
		arrAxisInG201[j] := 0;
	END_FOR
END_IF
(* **************************************************************************** *)

IF NOT gpCh[nChan]^.bahn_state.g201_active_r THEN
	IF CNCSystem.Channel[nChan].ActMode = HLI_IMCM_AUTOMATIC_MODE OR CNCSystem.Channel[nChan].ActMode = HLI_IMCM_MDI_MODE THEN
		nState := 0; 
	END_IF
END_IF

CASE nState OF
	0: (* IDLE *)
		bBusy := FALSE;
		bInManualMode := FALSE;

		IF (CNCSystem.Channel[nChan].ActMode = HLI_IMCM_MANUAL_MODE AND
    		stManualModeParameter.stChannelParameter.eManualType <> E_CNC_ManualType.NoManualMode AND
    		CNCSystem.Channel[nChan].ActState = HLI_IMCM_PROCESS_ACTIVE) OR  (* Manual Mode *)
   			((arrAxisinG201[0] <> 0)    (* mindestens eine Achse in G201 *) AND
    		((CNCSystem.Channel[nChan].ActState = HLI_IMCM_PROCESS_ACTIVE) OR
     		(CNCSystem.Channel[nChan].ActState = HLI_IMCM_PROCESS_HOLD))) (* Channel is active *)
		THEN			
			bError 		:= FALSE;
			nErrorID 	:= 0;

			stManualModeParameterOld     := stManualModeParameter;
			ActChannelModeOld   		:= cncsystem.Channel[nChan].ActMode;			
			i:= 0;
			nState := 10;

		END_IF

	10:		// Restore Manual State										
			FOR j := 0 TO HLI_KEY_MAXIDX DO
				IF (stManualModeControlElementState.stKeyUnit[j].nChan = nChan) THEN
					stManualModeControlElementState.stKeyUnit[j].nChan := -1;
					stManualModeControlElementState.stKeyUnit[j].nLogAxisId := 0;
					stManualModeControlElementState.stKeyUnit[j].nInputParameterIdx := -1;
				END_IF													
			END_FOR
			
			FOR j := 0 TO HLI_HW_MAXIDX DO
				IF (stManualModeControlElementState.stHWUnit[j].nChan = nChan) THEN
					stManualModeControlElementState.stHWUnit[j].nChan := -1;
					stManualModeControlElementState.stHWUnit[j].nLogAxisId := 0;
					stManualModeControlElementState.stHWUnit[j].nInputParameterIdx := -1;
				END_IF													
			END_FOR
	
			n:= 0;		
			nState := 20;						
			
20: 	// Deactivation 
		IF (n <= HLI_CH_AX_MAXIDX) THEN
			IF gpCh[nChan]^.bahn_state.coord_r[n].hb_display_r.control_element <> 0 THEN 
				IF NOT gpCh[nChan]^.hb_mc_control.activation.command_semaphor_rw THEN		
						gpCh[nChan]^.hb_mc_control.activation.command_w.log_achs_nr := gpCh[nChan]^.bahn_state.coord_r[n].log_achs_nr_r;
						gpCh[nChan]^.hb_mc_control.activation.command_w.control_element := 0;
						gpCh[nChan]^.hb_mc_control.activation.command_w.operation_mode := 0;
						
						IF (gpCh[nChan]^.bahn_state.coord_r[n].hb_display_r.operation_mode = 1) THEN
							stManualModeControlElementState.stHWUnit[gpCh[nChan]^.bahn_state.coord_r[n].hb_display_r.control_element-1].nChan := -1;
							stManualModeControlElementState.stHWUnit[gpCh[nChan]^.bahn_state.coord_r[n].hb_display_r.control_element-1].nLogAxisId :=0;
							stManualModeControlElementState.stHWUnit[gpCh[nChan]^.bahn_state.coord_r[n].hb_display_r.control_element-1].nInputParameterIdx := -1;	
						ELSE
							stManualModeControlElementState.stKeyUnit[gpCh[nChan]^.bahn_state.coord_r[n].hb_display_r.control_element-1].nChan := -1;
							stManualModeControlElementState.stKeyUnit[gpCh[nChan]^.bahn_state.coord_r[n].hb_display_r.control_element-1].nLogAxisId :=0;
							stManualModeControlElementState.stKeyUnit[gpCh[nChan]^.bahn_state.coord_r[n].hb_display_r.control_element-1].nInputParameterIdx := -1;						
						END_IF
						gpCh[nChan]^.hb_mc_control.activation.command_semaphor_rw := TRUE;
						nState := 21;					
				END_IF
			ELSE
				n := n + 1;
			END_IF				
		END_IF

		IF n >HLI_CH_AX_MAXIDX THEN
			nState := 26;
		END_IF
21: 
		IF 	NOT gpCh[nChan]^.hb_mc_control.activation.command_semaphor_rw THEN						
			n := n+1;
			nState := 20;
		END_IF
		
		IF n > HLI_CH_AX_MAXIDX THEN
			nState := 26;
		END_IF			
			
		
						
26:     IF gpCh[nChan]^.bahn_state.g201_active_r THEN // Bei G201 kann kein Init String übergeben werden
			nState := 30;		
		ELSIF NOT stCmdModesStates.stModes.Manual THEN
    		nState := 0;
		ELSE						
			strInitParameter := '$R$N';	 					
			(* Activation of an manual mode string *)
			IF stManualModeParameter.stChannelParameter.stManualOption.bTrafoActive THEN
				strInitParameter := CONCAT(	strInitParameter,'$R$N#TRAFO ON$R$N');
			END_IF
			
			IF stManualModeParameter.stChannelParameter.stManualOption.bEcsActive THEN
					strInitParameter := CONCAT(strInitParameter,'$R$N#ECS ON$R$N');
			END_IF
			
			IF stManualModeParameter.stChannelParameter.stManualOption.bCAXActive THEN
					strInitParameter := CONCAT(strInitParameter,'$R$N#CAX$R$N');
			END_IF
						
			strInitParameter := CONCAT(strInitParameter, stManualModeParameter.stChannelParameter.strInitParameter);
			
			strZeroOffset := '';
			CASE stManualModeParameter.stChannelParameter.stManualOption.eZeroOffset OF
				0: strZeroOffset := '$R$NG53';
				1: strZeroOffset := '$R$NG54';
				2: strZeroOffset := '$R$NG55';
				3: strZeroOffset := '$R$NG56';
				4: strZeroOffset := '$R$NG57';
				5: strZeroOffset := '$R$NG58';
				6: strZeroOffset := '$R$NG59';					
			ELSE
				strZeroOffset  := CONCAT(strZeroOffset, '$R$NG159 = ');
				strZeroOffset  := CONCAT(strZeroOffset, INT_TO_STRING(stManualModeParameter.stChannelParameter.stManualOption.eZeroOffset));						 							
			END_CASE
							
			strInitParameter := CONCAT(strInitParameter, strZeroOffset);								 		
			strInitParameter := CONCAT(strInitParameter,'$R$NG200');
	
		IF 	(strInitParameterOld <> strInitParameter) THEN 								  		  
				IF 	NOT gpCh[nChan]^.channel_mc_control.mode_and_state.command_semaphor_rw THEN
					gpCh[nCHan]^.channel_mc_control.mode_and_state.command_w.to_mode := HLI_IMCM_MANUAL_MODE ;
					gpCh[nCHan]^.channel_mc_control.mode_and_state.command_w.to_state := HLI_IMCM_PROCESS_SELECTED;
					gpCh[nCHan]^.channel_mc_control.mode_and_state.command_w.channel_number := INT_TO_UDINT(nChan+1);
					pString := ADR(gpCh[nCHan]^.channel_mc_control.mode_and_state.command_w.parameter);
					pString^ := '';
					gpCh[nChan]^.channel_mc_control.mode_and_state.command_semaphor_rw := TRUE;
					TON_TimeOut(in:= FALSE);
					nState := 27;
				END_IF
			ELSE
					i := 0;
					nState := 30;
			END_IF
		END_IF

27:		IF  NOT stCmdModesStates.stModes.Manual THEN
			nstate := 0; 
		ELSIF CNCSystem.Channel[nChan].ActState = HLI_IMCM_PROCESS_SELECTED AND
			gpCh[nCHan]^.channel_mc_control.mode_and_state.command_semaphor_rw = FALSE
		THEN									
				gpCh[nCHan]^.channel_mc_control.mode_and_state.command_w.to_mode := HLI_IMCM_MANUAL_MODE ;
				gpCh[nCHan]^.channel_mc_control.mode_and_state.command_w.to_state := HLI_IMCM_PROCESS_ACTIVE;
				gpCh[nCHan]^.channel_mc_control.mode_and_state.command_w.channel_number := INT_TO_UDINT(nChan+1);
				pString := ADR(gpCh[nCHan]^.channel_mc_control.mode_and_state.command_w.parameter);			
				pString^ := strInitParameter;
				gpCh[nCHan]^.channel_mc_control.mode_and_state.command_semaphor_rw := TRUE;		
				TON_TimeOut(in:= FALSE);		
				nState := 28;			
		END_IF

		TON_TimeOut(in:=TRUE, PT:=T#5s);
		IF TON_TimeOut.Q THEN
			nState := 99;
		END_IF

28:		IF  NOT stCmdModesStates.stModes.Manual OR 
			CNCSystem.Channel[nChan].ActMode <> HLI_IMCM_MANUAL_MODE OR
			CNCSystem.Channel[nChan].ActState = HLI_IMCM_PROCESS_ERROR
		THEN 
			nState := 0;
		ELSIF (gpCh[nCHan]^.channel_mc_control.mode_and_state.command_semaphor_rw = FALSE)  AND
			CNCSystem.Channel[nChan].ActState = HLI_IMCM_PROCESS_ACTIVE 
			THEN														
				strInitParameterOld := strInitParameter;
				ManualActivation(bExecute := FALSE, 
								stManualModeControlElements := stManualModeControlElements ,
								stManualModeControlElementState:= stManualModeControlElementState);
				i := 0;
				IF (gpCh[nChan]^.bahn_state.g200_active_r) THEN	
					nState := 30;
				END_IF
						
		END_IF				
	
30: 	(* --- activate KeyControlUnits --- *)
		IF NOT stCmdModesStates.stModes.Manual AND NOT gpCh[nChan]^.bahn_state.g201_active_r THEN
			nState := 0;							
		ELSE							
			ManualActivation(bExecute := TRUE,
									nChan 			 := nChan,
									eManualType 	 := stManualModeParameter.stChannelParameter.eManualType,									
									stManualModeControlElementState:= stManualModeControlElementState,
									stManualModeControlElements := stManualModeControlElements,
									nInputParameterIdx := i,
									nHBA_Res 		 := stManualModeParameter.stChannelParameter.nHandwheelResolution,
									Inc 		     := stManualModeParameter.stChannelParameter.nInc,
									Speed 			 := stManualModeParameter.stAxisParameter.stControlUnit[i].nSpeed, // geändert alt nControlUnit
									nLogAxisNr 		 := stManualModeParameter.stAxisParameter.stControlUnit[i].nLogAxisNr); // geändert alt nControlUnit
			nState := 35;
		END_IF				
															
35: 	(* waiting for acknowledge *)
		ManualActivation(bExecute := FALSE, 
						stManualModeControlElements := stManualModeControlElements,
						stManualModeControlElementState:= stManualModeControlElementState);
		
		IF ManualActivation.bBusy = FALSE THEN
			IF ManualActivation.bError THEN
				nErrorId := ErrID_1;
				nState := 99;
			ELSE
				IF stManualModeParameter.stAxisParameter.stControlUnit[i+1].nLogAxisNr = 0 THEN
					i:=-1; (* reset the array counter *)				
					nState := 40;
				ELSE
					ManualActivation(bExecute := FALSE, 
									 stManualModeControlElements := stManualModeControlElements,
									 stManualModeControlElementState:= stManualModeControlElementState);
					nState := 30;
					i:= i+1;
				END_IF
			END_IF
		END_IF

40: 	(* endlich Handbetrieb *)
		bInManualMode := TRUE;
		
		IF (stManualModeParameter.stChannelParameter.eManualType <> E_CNC_ManualType.Handwheel) THEN
			FOR j := 0 TO HLI_KEY_MAXIDX DO
				IF stManualModeControlElementState.stKeyUnit[j].nChan = nChan AND stManualModeControlElementState.stKeyUnit[j].nLogAxisId <> 0 THEN				
					ManualExecution[j](	nChan := nChan,
									nKeyControlUnit := j,
									bKeyPos := stManualModeControlElements.stControlKeys[stManualModeControlElementState.stKeyUnit[j].nInputParameterIdx].bKeyPos,					// geändert 	nControlUnit
									bKeyNeg := stManualModeControlElements.stControlKeys[stManualModeControlElementState.stKeyUnit[j].nInputParameterIdx].bKeyNeg); (* no timeouts *)
									
					ManualExecutionRapidMode[j](nChan := nChan,
									nKeyControlUnit := j,
									bExecute := stManualModeControlElements.stControlKeys[stManualModeControlElementState.stKeyUnit[j].nInputParameterIdx].bKeyRapid); (* no timeouts *)
				END_IF
			END_FOR			
		ELSE				
			(* Handradincremente werden immer vom ersten Kanal entgegen genommen*)
			FOR j := 0 TO HLI_HW_MAXIDX DO
				IF (stManualModeControlElementState.stHWUnit[j].nChan = nChan AND stManualModeControlElementState.stHWUnit[j].nLogAxisId <>  0)  THEN 
					gpCh[0]^.hb_mc_control.handwheel_incs[j].command_w := stManualModeControlElements.nHandwheelInc[stManualModeControlElementState.stHWUnit[j].nInputParameterIdx];
				END_IF			
			END_FOR
		END_IF

		(* end of manual mode *)
		 IF (bManual = FALSE) OR                                                                                                             
         	MEMCMP(ADR(stManualModeParameter),ADR(stManualModeParameterOld),SIZEOF(stManualModeParameter)-SIZEOF(stManualModeParameter.stChannelParameter.strInitParameter))<>0 OR                                                      
            stManualModeParameter.stChannelParameter.strInitParameter <> stManualModeParameterOld.stChannelParameter.strInitParameter OR                                                          
            cncsystem.Channel[nChan].ActMode <> ActChannelModeOld OR                                       
            (CNCSystem.Channel[nChan].ActMode =  HLI_IMCM_MANUAL_MODE AND CNCSystem.Channel[nChan].ActState <> HLI_IMCM_PROCESS_ACTIVE) OR                                                   
            stManualModeParameter.stChannelParameter.eManualType = E_CNC_ManualType.NoManualMode
            THEN
		
				FOR j := 0 TO HLI_KEY_MAXIDX DO
					IF stManualModeControlElementState.stKeyUnit[j].nChan = nChan THEN
						ManualExecution[j](nChan := nChan,	nKeyControlUnit := j, bKeyPos := FALSE, bKeyNeg := FALSE); (* no timeouts *)		
					END_IF		
				END_FOR
						
				i:=1 (* resets the counter for the following deactivation *);			

				stManualModeParameterOld 	:= stManualModeParameter;
	
				IF cncsystem.Channel[nChan].ActMode <> ActChannelModeOld OR stManualModeParameter.stChannelParameter.eManualType = E_CNC_ManualType.NoManualMode THEN
					ActChannelModeOld := cncsystem.Channel[nChan].ActMode;			
					nState := 0;
				ELSE
					nState := 0; (* evt. wird hier auch eine Verzoegerungszeit benötigt,
										  Fehler 150054 dann nState = 0 *)
					bInManualMode := FALSE;
				END_IF
		END_IF

99: 	(* error handling *)	
		bBusy := FALSE;
		bError := TRUE;
		
		(* end of manual mode *)
			IF NOT gpCh[nCHan]^.channel_mc_control.mode_and_state.command_semaphor_rw AND 
			CNCSystem.Channel[nChan].ActState <>  HLI_IMCM_PROCESS_ERROR
			THEN;
				gpCh[nCHan]^.channel_mc_control.mode_and_state.command_w.to_mode := HLI_IMCM_MANUAL_MODE ;
				gpCh[nCHan]^.channel_mc_control.mode_and_state.command_w.to_state := HLI_IMCM_PROCESS_ERROR;
				gpCh[nCHan]^.channel_mc_control.mode_and_state.command_w.channel_number := INT_TO_UDINT(nChan+1);			
				gpCh[nCHan]^.channel_mc_control.mode_and_state.command_semaphor_rw := TRUE;	
			END_IF
			nState := 0;
		
		(* end of manual mode *)
		IF bManual = FALSE THEN
			bBusy := FALSE;
			nState := 0;
		END_IF

END_CASE

END_FUNCTION_BLOCK

// CNC/2 OperationMode/ModeManual/PRG_AnalogJoystick
PROGRAM PRG_AnalogJoystick
VAR_INPUT
	nLogAxisNr: UINT;
	/// Actual Analog Value 
	Analog_Value: DINT;
	/// static signal : Analog Min Value 
	AnalogValueMin: DINT;
	/// static signal : Analog Max Value 
	AnalogValueMax: DINT;
	/// Dead Band for Zero Value 
	AnalogValueZeroDeadBand: DINT;
END_VAR
VAR_IN_OUT
	bKeyPos: BOOL;
	bKeyNeg: BOOL;
END_VAR
VAR
	/// Index of axis specific HLI area 
	nHliAxisIdx: INT;
	Norm_AnalogValue: LREAL;
	Zero_AnalogValue: LREAL;
	Override: LREAL;
END_VAR

(* ========================================================= *)
(*    Prog: Analog JoyStick			                  		 *)
(* --------------------------------------------------------- *)
(*   Desc:                                                   *)
(*   Author: TV	, MiB	                                         *)
(*   Date: 24.07.2015                                       *)
(*   Rev.: 6.0                                               *)
(* ========================================================= *)
	Norm_AnalogValue := (AnalogValueMax - AnalogValueMin);
	Zero_AnalogValue := AnalogValueMin + Norm_AnalogValue / 2;

	IF nLogAxisNr > 0 AND Norm_AnalogValue > 0 THEN
		nHliAxisIdx :=  HLI3_GetHliAxisIdx(UINT_TO_INT(nLogAxisNr));
		IF (nHliAxisIdx = -1) THEN
			RETURN;
		END_IF
		gpAx[nHliAxisIdx]^.ipo_mc_control.override.enable_w := TRUE;
		gpAx[nHliAxisIdx]^.ipo_mc_control.override_valid.enable_w := TRUE;
		gpAx[nHliAxisIdx]^.ipo_mc_control.override_valid.command_w := TRUE;
		Override := ABS(((Analog_Value  - AnalogValueMin) * 200 / Norm_AnalogValue)-100);

		IF Override > 100.0 THEN Override := 100.0; END_IF

		IF Analog_Value > Zero_AnalogValue THEN bKeyPos := TRUE; bKeyNeg := FALSE; ELSE bKeyPos := FALSE; END_IF
		IF Analog_Value < Zero_AnalogValue THEN bKeyNeg := TRUE; bKeyPos := FALSE; ELSE bKeyNeg := FALSE; END_IF

		IF Analog_Value > (Zero_AnalogValue - AnalogValueZeroDeadBand) AND Analog_Value < (Zero_AnalogValue + AnalogValueZeroDeadBand) THEN
			Override := 0;
			bKeyNeg := FALSE;
			bKeyPos := FALSE;
		END_IF

		gpAx[nHliAxisIdx]^.ipo_mc_control.override.command_w := LREAL_TO_UINT(Override * 10);
	END_IF

END_PROGRAM

// CNC/8 Mis/HLI3_GetHliAxisIdx
FUNCTION HLI3_GetHliAxisIdx : INT
VAR_INPUT
	nLogAxisId: INT;
END_VAR
VAR
	i: INT;
END_VAR

(* ========================================================= *)
(*    FUN: HLI3_GetHliAxisIdx                            *)
(* --------------------------------------------------------- *)
(*   Desc: returns teh HliAxisIdx for a given logical Axis id      	*)
(*   Author: MiB                                             *)
(*   Date: 19.11.2012                                        *)
(*   Rev.: 1.0                                               *)
(* ========================================================= *)
HLI3_GetHliAxisIdx := -1;
FOR i := 0 TO UDINT_TO_INT(gNrAx) DO
	IF nLogAxisId = UINT_TO_INT(gpAx[i]^.head.log_ax_nr_r) THEN
		HLI3_GetHliAxisIdx := i;
		RETURN;
	END_IF
END_FOR

END_FUNCTION

// CNC/3 Control/HLI3_SetAxisOverride
FUNCTION HLI3_SetAxisOverride : BOOL
VAR_INPUT
	/// number of Axis 
	nHliAxisIdx: INT;
	nOverride: UINT;
END_VAR

(* ========================================================= *)
(*    FUN: HLI_SetAxisOverride                               *)
(* --------------------------------------------------------- *)
(*   Desc: Set the Axis Override                             *)
(* Author: TV                                                *)
(*   Date: 20.12.2007                                        *)
(*   Rev.: 1.0                                               *)
(*   Rev.: 1.1 MiB 19.11.2012 Tc3                            *)
(* ========================================================= *)
IF NOT (HLI3_CheckAxisValid(nHliAxisIdx := nHliAxisIdx)) THEN
	HLI3_SetAxisOverride := FALSE;
	RETURN;
END_IF


(* Limit the override *)
IF nOverride > 1200	THEN nOverride := 1200; END_IF
IF nOverride < 0 THEN nOverride := 0; END_IF

	gpAx[nHliAxisIdx]^.ipo_mc_control.override.enable_w  := TRUE;
	gpAx[nHliAxisIdx]^.ipo_mc_control.override.command_w := nOverride;

HLI3_SetAxisOverride := TRUE;

END_FUNCTION

// CNC/2 OperationMode/HLI3_AxisReset
FUNCTION HLI3_AxisReset : BOOL
VAR_INPUT
	/// Channel number 
	nChanNo: INT;
	/// Axis number 
	nHliAxisIdx: INT;
END_VAR
VAR
	/// local pointer to data of actual axis 
	pAxisData: POINTER TO HIGH_LEVEL_INTERFACE_AX;
END_VAR

(* ========================================================= *)
(*    FUN: HLI3_QuitAxisReset                                 *)
(* --------------------------------------------------------- *)
(*   Desc:                                                   *)
(* Author: MK , MiB                                          *)
(*   Date: 20.11.2012                                        *)
(*   Rev.: 1.1                                               *)
(* ========================================================= *)


HLI3_AxisReset := FALSE;
IF NOT HLI3_CheckAxisValid(nHliAxisIdx := nHliAxisIdx) THEN
	RETURN;
END_IF

IF gpAx[nHliAxisIdx] = 0 THEN
	RETURN;
END_IF


(* get pointer to axis data *)
pAxisData := gpAx[nHliAxisIdx];
IF pAxisData^.ipo_state.cnc_channel_r = INT_TO_UINT(nChanNo) THEN (* it's an axis of the channel *)
	(* is a reset commanded *)
	IF pAxisData^.ipo_lc_control.plc_reset.command_r = TRUE THEN
		(* quit this reset *)
		pAxisData^.ipo_lc_control.plc_reset.state_w := TRUE;	
		HLI3_AxisReset := TRUE;
	END_IF
END_IF

END_FUNCTION

// CNC/2 OperationMode/HLI3_ChannelModeAuto
FUNCTION HLI3_ChannelModeAuto : BOOL
VAR_INPUT	
	nChanIdx: INT;
	ProgramName: STRING(HLI_IMCM_MODE_STATE_PARAM_STRL);			
END_VAR
VAR_IN_OUT
	stCmdModesStates    : ST_CNCCmdModesStates;	
END_VAR
VAR
	pString: POINTER TO STRING(HLI_IMCM_MODE_STATE_PARAM_STRL);
END_VAR

(* ========================================================= *)
(*    FUN: HLI_ChannelModeAuto                               *)
(* --------------------------------------------------------- *)
(*   Desc: switch channel to Automatic mode / xxx            *)
(*   Author: MK,MiB, TV                                      *)
(*   Date: 03.03.2017                                        *)
(*   Rev.: 1.5                                               *)
(* ========================================================= *)

IF (NOT gpCh[nChanIdx]^.channel_mc_control.mode_and_state.command_semaphor_rw) THEN    (* only if semaphor is FALSE...... *)
	IF stCmdModesStates.stStates.Selected THEN
		stCmdModesStates.stStates.Selected := FALSE;
		gpCh[nChanIdx]^.channel_mc_control.mode_and_state.command_w.to_mode := HLI_IMCM_AUTOMATIC_MODE;
		gpCh[nChanIdx]^.channel_mc_control.mode_and_state.command_w.to_state := HLI_IMCM_PROCESS_SELECTED;	
		pString := ADR(gpCh[nChanIdx]^.channel_mc_control.mode_and_state.command_w.parameter);			
		pString^ := ProgramName;				
		gpCh[nChanIdx]^.channel_mc_control.mode_and_state.command_semaphor_rw  := TRUE;		
	END_IF
	
	IF stCmdModesStates.stStates.Ready THEN
		stCmdModesStates.stStates.Ready := FALSE;
		gpCh[nChanIdx]^.channel_mc_control.mode_and_state.command_w.to_mode := HLI_IMCM_AUTOMATIC_MODE;
		gpCh[nChanIdx]^.channel_mc_control.mode_and_state.command_w.to_state := HLI_IMCM_PROCESS_READY;		
		pString := ADR(gpCh[nChanIdx]^.channel_mc_control.mode_and_state.command_w.parameter);			
		pString^ := ProgramName;				
		gpCh[nChanIdx]^.channel_mc_control.mode_and_state.command_semaphor_rw  := TRUE;		
	END_IF
	
	IF stCmdModesStates.stStates.Active THEN
		stCmdModesStates.stStates.Active := FALSE;
		gpCh[nChanIdx]^.channel_mc_control.mode_and_state.command_w.to_mode := HLI_IMCM_AUTOMATIC_MODE;
		gpCh[nChanIdx]^.channel_mc_control.mode_and_state.command_w.to_state := HLI_IMCM_PROCESS_ACTIVE;		
		pString := ADR(gpCh[nChanIdx]^.channel_mc_control.mode_and_state.command_w.parameter);			
		pString^ := ProgramName;				
		gpCh[nChanIdx]^.channel_mc_control.mode_and_state.command_semaphor_rw  := TRUE;		
	END_IF
	
	IF stCmdModesStates.stStates.Hold THEN
		stCmdModesStates.stStates.Hold:= FALSE;
		gpCh[nChanIdx]^.channel_mc_control.mode_and_state.command_w.to_mode:= HLI_IMCM_AUTOMATIC_MODE;
		gpCh[nChanIdx]^.channel_mc_control.mode_and_state.command_w.to_state := HLI_IMCM_PROCESS_HOLD;		
		gpCh[nChanIdx]^.channel_mc_control.mode_and_state.command_semaphor_rw  := TRUE;
	END_IF
	
	IF stCmdModesStates.stStates.Reset THEN
		stCmdModesStates.stStates.Reset := FALSE;
		gpCh[nChanIdx]^.channel_mc_control.mode_and_state.command_w.to_mode := HLI_IMCM_AUTOMATIC_MODE;
		gpCh[nChanIdx]^.channel_mc_control.mode_and_state.command_w.to_state:= HLI_IMCM_PROCESS_RESETTING;		
		gpCh[nChanIdx]^.channel_mc_control.mode_and_state.command_semaphor_rw  := TRUE;		
	END_IF
	
	HLI3_ChannelModeAuto := TRUE;
ELSE
	HLI3_ChannelModeAuto := FALSE;
END_IF

END_FUNCTION

// CNC/2 OperationMode/HLI3_ChannelModeManual
FUNCTION HLI3_ChannelModeManual : BOOL
VAR_INPUT	
	nChanIdx: INT;	
END_VAR

VAR_IN_OUT
	stCmdModesStates    : ST_CNCCmdModesStates;	
END_VAR

VAR
	pString: POINTER TO STRING;
END_VAR

(* ========================================================= *)
(*    FUN: HLI_ChannelModeManual                             *)
(* --------------------------------------------------------- *)
(*   Desc: switch channel to Manual mode / xxx               *)
(*   Author: MK, MiB, TV, RCH                                *)
(*   Date: 03.03.2017                                        *)
(*   Rev.: 1.5                                               *)
(* ========================================================= *)

IF (NOT  gpCh[nChanIdx]^.channel_mc_control.mode_and_state.command_semaphor_rw) THEN    (* only if semaphor is FALSE...... *)
	IF stCmdModesStates.stStates.Selected THEN
		stCmdModesStates.stStates.Selected := FALSE;
		gpCh[nChanIdx]^.channel_mc_control.mode_and_state.command_w.to_mode := HLI_IMCM_MANUAL_MODE;
		gpCh[nChanIdx]^.channel_mc_control.mode_and_state.command_w.to_state := HLI_IMCM_PROCESS_SELECTED;		
		pString := ADR(gpCh[nChanIdx]^.channel_mc_control.mode_and_state.command_w.parameter);			
		pString^ := '';	
		gpCh[nChanIdx]^.channel_mc_control.mode_and_state.command_semaphor_rw := TRUE;		
	END_IF
	
	IF stCmdModesStates.stStates.Ready THEN
		stCmdModesStates.stStates.Ready := FALSE;
		gpCh[nChanIdx]^.channel_mc_control.mode_and_state.command_w.to_mode := HLI_IMCM_MANUAL_MODE;
		gpCh[nChanIdx]^.channel_mc_control.mode_and_state.command_w.to_state := HLI_IMCM_PROCESS_READY;		
		pString := ADR(gpCh[nChanIdx]^.channel_mc_control.mode_and_state.command_w.parameter);			
		pString^ := '';
		gpCh[nChanIdx]^.channel_mc_control.mode_and_state.command_semaphor_rw := TRUE;		
	END_IF
	
	IF stCmdModesStates.stStates.Active THEN
		stCmdModesStates.stStates.Active := FALSE;
		gpCh[nChanIdx]^.channel_mc_control.mode_and_state.command_w.to_mode := HLI_IMCM_MANUAL_MODE;
		gpCh[nChanIdx]^.channel_mc_control.mode_and_state.command_w.to_state := HLI_IMCM_PROCESS_ACTIVE;		
		pString := ADR(gpCh[nChanIdx]^.channel_mc_control.mode_and_state.command_w.parameter);			
		pString^ := '';						
		gpCh[nChanIdx]^.channel_mc_control.mode_and_state.command_semaphor_rw := TRUE;	
	END_IF
	
	IF stCmdModesStates.stStates.Hold THEN
		stCmdModesStates.stStates.Hold := FALSE;
		gpCh[nChanIdx]^.channel_mc_control.mode_and_state.command_w.to_mode := HLI_IMCM_MANUAL_MODE;
		gpCh[nChanIdx]^.channel_mc_control.mode_and_state.command_w.to_state := HLI_IMCM_PROCESS_HOLD;		
		gpCh[nChanIdx]^.channel_mc_control.mode_and_state.command_semaphor_rw := TRUE;		
	END_IF
	
	IF stCmdModesStates.stStates.Reset THEN
		stCmdModesStates.stStates.Reset := FALSE;
		gpCh[nChanIdx]^.channel_mc_control.mode_and_state.command_w.to_mode:= HLI_IMCM_MANUAL_MODE;
		gpCh[nChanIdx]^.channel_mc_control.mode_and_state.command_w.to_state := HLI_IMCM_PROCESS_RESETTING;		
		gpCh[nChanIdx]^.channel_mc_control.mode_and_state.command_semaphor_rw:= TRUE;		
	END_IF

	HLI3_ChannelModeManual := TRUE;
ELSE
	HLI3_ChannelModeManual := FALSE;
END_IF

END_FUNCTION

// CNC/2 OperationMode/HLI3_ChannelModeMDI
FUNCTION HLI3_ChannelModeMDI : BOOL
VAR_INPUT	
	nChanIdx: INT;	
	/// pointer to the MDI program string 
	pMDIString: POINTER TO STRING(HLI_IMCM_MODE_STATE_PARAM_STRL);
END_VAR

VAR_IN_OUT
	stCmdModesStates    : ST_CNCCmdModesStates;	
END_VAR
VAR
	pString: POINTER TO STRING(HLI_IMCM_MODE_STATE_PARAM_STRL);
END_VAR

(* ========================================================= *)
(*    FUN: HLI_ChannelModeMDI                                *)
(* --------------------------------------------------------- *)
(*   Desc: switch channel to MDI mode / xxx                  *)
(*   Author: MK, TV, MiB, Rch                                *)
(*   Date: 18.07.2002                                        *)
(*   Last: 03.03.2017                      				     *)
(*   Rev.: 1.7                                               *)
(* ========================================================= *)

IF (NOT gpCh[nChanIdx]^.channel_mc_control.mode_and_state.command_semaphor_rw) THEN  (* only if semaphor is FALSE...... *)

	IF stCmdModesStates.stStates.Selected THEN
		stCmdModesStates.stStates.Selected := FALSE;
		gpCh[nChanIdx]^.channel_mc_control.mode_and_state.command_w.to_mode := HLI_IMCM_MDI_MODE;
		gpCh[nChanIdx]^.channel_mc_control.mode_and_state.command_w.to_state := HLI_IMCM_PROCESS_SELECTED;
		pString := ADR(gpCh[nChanIdx]^.channel_mc_control.mode_and_state.command_w.parameter);					
		pString^ := pMDIString^;
		gpCh[nChanIdx]^.channel_mc_control.mode_and_state.command_semaphor_rw := TRUE;		
	END_IF
	
	IF stCmdModesStates.stStates.Ready THEN
		stCmdModesStates.stStates.Ready := FALSE;
		gpCh[nChanIdx]^.channel_mc_control.mode_and_state.command_w.to_mode:= HLI_IMCM_MDI_MODE;
		gpCh[nChanIdx]^.channel_mc_control.mode_and_state.command_w.to_state := HLI_IMCM_PROCESS_READY;		
		gpCh[nChanIdx]^.channel_mc_control.mode_and_state.command_semaphor_rw := TRUE;		
	END_IF
	
	IF stCmdModesStates.stStates.Active THEN
		stCmdModesStates.stStates.Active := FALSE;
		gpCh[nChanIdx]^.channel_mc_control.mode_and_state.command_w.to_mode := HLI_IMCM_MDI_MODE;
		gpCh[nChanIdx]^.channel_mc_control.mode_and_state.command_w.to_state := HLI_IMCM_PROCESS_ACTIVE;
		pString := ADR(gpCh[nChanIdx]^.channel_mc_control.mode_and_state.command_w.parameter);					
		pString^ := pMDIString^;
		gpCh[nChanIdx]^.channel_mc_control.mode_and_state.command_semaphor_rw := TRUE;		
	END_IF
	
	IF stCmdModesStates.stStates.Hold THEN
		stCmdModesStates.stStates.Hold := FALSE;
		gpCh[nChanIdx]^.channel_mc_control.mode_and_state.command_w.to_mode := HLI_IMCM_MDI_MODE;
		gpCh[nChanIdx]^.channel_mc_control.mode_and_state.command_w.to_state:= HLI_IMCM_PROCESS_HOLD;		
		gpCh[nChanIdx]^.channel_mc_control.mode_and_state.command_semaphor_rw := TRUE;		
	END_IF
	
	IF stCmdModesStates.stStates.Reset THEN
		stCmdModesStates.stStates.Reset := FALSE;
		gpCh[nChanIdx]^.channel_mc_control.mode_and_state.command_w.to_mode := HLI_IMCM_MDI_MODE;
		gpCh[nChanIdx]^.channel_mc_control.mode_and_state.command_w.to_state := HLI_IMCM_PROCESS_RESETTING;		
		gpCh[nChanIdx]^.channel_mc_control.mode_and_state.command_semaphor_rw := TRUE;		
	END_IF
	HLI3_ChannelModeMDI := TRUE;	
ELSE
	HLI3_ChannelModeMDI := FALSE;
END_IF

END_FUNCTION

// CNC/2 OperationMode/HLI3_ChannelModeReference
FUNCTION HLI3_ChannelModeReference : BOOL
VAR_INPUT	
	nChanIdx: INT;	
	/// the referencing string 
	sRefPosString: STRING(HLI_IMCM_MODE_STATE_PARAM_STRL);	
END_VAR

VAR_IN_OUT
	stCmdModesStates    : ST_CNCCmdModesStates;	
END_VAR

VAR
	pString: POINTER TO STRING(HLI_IMCM_MODE_STATE_PARAM_STRL);
END_VAR

